SPLINE
SPL {X  -131.598, Y  +769.376, Z    +0.000, E1   -56.871, E3 +79450.846}
SPL {X  -152.760, Y  +729.846, Z    +0.000, E1   -44.713, E3 +79457.898}
SPL {X  -158.868, Y  +709.157, Z    +0.000, E1   -33.466, E3 +79459.099}
SPL {X  -161.987, Y  +689.949, Z    +0.000, E1   -18.777, E3 +79460.061}
SPL {X  -162.803, Y  +675.860, Z    +0.000, E1    -4.958, E3 +79460.043}
SPL {X  -162.820, Y  +671.500, Z    +0.000, E1    +0.000, E3 +79459.579}
SPL {X  -162.820, Y  +669.410, Z    +0.000, E1    +4.515, E3 +79459.341}
SPL {X  -162.820, Y  +664.781, Z    +0.000, E1   +16.411, E3 +79459.337}
SPL {X  -162.820, Y  +659.650, Z    +0.000, E1   +29.778, E3 +79459.346}
SPL {X  -162.820, Y  +654.031, Z    +0.000, E1   +42.449, E3 +79459.260}
SPL {X  -162.820, Y  +647.611, Z    +0.000, E1   +52.483, E3 +79459.791}
SPL {X  -162.820, Y  +637.134, Z    +0.000, E1   +65.232, E3 +79458.039}
SPL {X  -162.820, Y  +616.721, Z    +0.000, E1   +72.273, E3 +79461.773}
SPL {X  -162.820, Y  +577.172, Z    +0.000, E1   +75.843, E3 +79471.753}
SPL {X  -159.895, Y  +349.775, Z    +0.000, E1   +76.042, E3 +79563.419}
ENDSPLINE

SPLINE
SPL {X  -160.357, Y  +352.285, Z    +0.000, E1   +74.783, E3 +79576.357}
ENDSPLINE

SPLINE
SPL {X  -145.737, Y  +307.897, Z    +0.000, E1   +77.368, E3 +79568.932}
SPL {X  -145.329, Y  +307.084, Z    +0.000, E1   +76.571, E3 +79577.768}
ENDSPLINE

SPLINE
SPL {X  -145.355, Y  +307.136, Z    +0.000, E1   +75.607, E3 +79587.292}
ENDSPLINE

SPLINE
SPL {X  -144.515, Y  +305.495, Z    +0.000, E1   +74.543, E3 +79598.101}
SPL {X  -143.690, Y  +303.925, Z    +0.000, E1   +73.372, E3 +79608.840}
SPL {X  -141.993, Y  +300.823, Z    +0.000, E1   +72.659, E3 +79616.265}
SPL {X  -138.166, Y  +294.358, Z    +0.000, E1   +72.281, E3 +79622.726}
SPL {X  -134.385, Y  +288.571, Z    +0.000, E1   +71.826, E3 +79628.990}
SPL {X  -130.773, Y  +283.501, Z    +0.000, E1   +71.398, E3 +79634.414}
SPL {X  -126.922, Y  +278.513, Z    +0.000, E1   +70.767, E3 +79640.568}
SPL {X  -123.520, Y  +274.419, Z    +0.000, E1   +70.342, E3 +79644.767}
SPL {X  -117.513, Y  +267.801, Z    +0.000, E1   +72.197, E3 +79641.115}
SPL {X   -63.140, Y  +230.421, Z    +0.000, E1   +55.875, E3 +79810.554}
ENDSPLINE

SPLINE
SPL {X  -130.329, Y  +282.905, Z    +0.000, E1   +55.659, E3 +79968.890}
SPL {X  -154.728, Y  +329.807, Z    +0.000, E1   +40.640, E3 +79978.271}
SPL {X  -160.994, Y  +356.185, Z    +0.000, E1   +24.373, E3 +79980.864}
SPL {X  -162.637, Y  +372.778, Z    +0.000, E1   +10.098, E3 +79980.884}
SPL {X  -162.820, Y  +382.419, Z    +0.000, E1    +0.163, E3 +79980.444}
SPL {X  -162.820, Y  +383.794, Z    +0.000, E1    -2.626, E3 +79980.162}
SPL {X  -162.820, Y  +387.647, Z    +0.000, E1   -11.488, E3 +79980.166}
SPL {X  -162.820, Y  +394.732, Z    +0.000, E1   -28.992, E3 +79980.084}
SPL {X  -162.820, Y  +403.075, Z    +0.000, E1   -46.096, E3 +79980.314}
SPL {X  -162.820, Y  +414.705, Z    +0.000, E1   -61.052, E3 +79979.760}
SPL {X  -162.820, Y  +466.149, Z    +0.000, E1   -74.732, E3 +79989.756}
SPL {X  -160.066, Y  +703.318, Z    +0.000, E1   -76.774, E3 +80074.603}
ENDSPLINE

SPLINE
SPL {X  -161.105, Y  +697.069, Z    +0.000, E1   -74.557, E3 +80096.218}
ENDSPLINE

SPLINE
SPL {X  -159.270, Y  +707.314, Z    +0.000, E1   -74.359, E3 +80104.241}
SPL {X  -156.868, Y  +717.123, Z    +0.000, E1   -74.182, E3 +80111.747}
SPL {X  -153.226, Y  +728.564, Z    +0.000, E1   -73.755, E3 +80122.756}
SPL {X  -149.090, Y  +738.941, Z    +0.000, E1   -73.348, E3 +80132.329}
SPL {X  -145.714, Y  +746.149, Z    +0.000, E1   -72.951, E3 +80139.916}
SPL {X  -142.592, Y  +752.100, Z    +0.000, E1   -72.554, E3 +80146.449}
SPL {X  -139.608, Y  +757.285, Z    +0.000, E1   -72.326, E3 +80151.118}
SPL {X  -136.902, Y  +761.638, Z    +0.000, E1   -71.857, E3 +80156.886}
SPL {X  -133.350, Y  +766.925, Z    +0.000, E1   -71.498, E3 +80162.206}
SPL {X  -129.687, Y  +771.946, Z    +0.000, E1   -71.061, E3 +80167.572}
SPL {X  -126.374, Y  +776.164, Z    +0.000, E1   -70.494, E3 +80172.826}
SPL {X  -123.763, Y  +779.297, Z    +0.000, E1   -70.128, E3 +80176.201}
SPL {X  -119.350, Y  +784.252, Z    +0.000, E1   -71.016, E3 +80175.402}
SPL {X   -61.593, Y  +824.220, Z    +0.000, E1   -55.970, E3 +80341.717}
ENDSPLINE

SPLINE
SPL {X  -131.598, Y  +769.376, Z    +0.000, E1   -56.871, E3 +80507.989}
SPL {X  -152.760, Y  +729.846, Z    +0.000, E1   -44.713, E3 +80515.041}
SPL {X  -159.952, Y  +703.925, Z    +0.000, E1   -29.977, E3 +80516.544}
SPL {X  -162.596, Y  +682.036, Z    +0.000, E1   -11.376, E3 +80517.264}
SPL {X  -162.820, Y  +671.380, Z    +0.000, E1    +0.035, E3 +80516.703}
SPL {X  -162.820, Y  +668.318, Z    +0.000, E1    +7.404, E3 +80516.440}
SPL {X  -162.820, Y  +664.781, Z    +0.000, E1   +16.411, E3 +80516.480}
SPL {X  -162.820, Y  +659.650, Z    +0.000, E1   +29.778, E3 +80516.489}
SPL {X  -162.820, Y  +651.175, Z    +0.000, E1   +47.162, E3 +80516.639}
SPL {X  -162.820, Y  +633.243, Z    +0.000, E1   +67.111, E3 +80515.894}
SPL {X  -162.820, Y  +577.172, Z    +0.000, E1   +75.843, E3 +80528.896}
SPL {X  -159.895, Y  +349.775, Z    +0.000, E1   +76.042, E3 +80620.562}
ENDSPLINE

SPLINE
SPL {X  -160.357, Y  +352.285, Z    +0.000, E1   +74.783, E3 +80633.500}
ENDSPLINE

SPLINE
SPL {X  -145.737, Y  +307.897, Z    +0.000, E1   +77.368, E3 +80626.075}
SPL {X  -145.329, Y  +307.084, Z    +0.000, E1   +76.571, E3 +80634.911}
ENDSPLINE

SPLINE
SPL {X  -145.355, Y  +307.136, Z    +0.000, E1   +75.607, E3 +80644.435}
ENDSPLINE

SPLINE
SPL {X  -144.515, Y  +305.495, Z    +0.000, E1   +74.543, E3 +80655.244}
SPL {X  -143.690, Y  +303.925, Z    +0.000, E1   +73.372, E3 +80665.983}
SPL {X  -141.993, Y  +300.823, Z    +0.000, E1   +72.659, E3 +80673.408}
SPL {X  -138.166, Y  +294.358, Z    +0.000, E1   +72.281, E3 +80679.869}
SPL {X  -134.385, Y  +288.571, Z    +0.000, E1   +71.826, E3 +80686.132}
SPL {X  -130.773, Y  +283.501, Z    +0.000, E1   +71.398, E3 +80691.557}
SPL {X  -126.922, Y  +278.513, Z    +0.000, E1   +70.767, E3 +80697.711}
SPL {X  -123.520, Y  +274.419, Z    +0.000, E1   +70.342, E3 +80701.909}
SPL {X  -117.513, Y  +267.801, Z    +0.000, E1   +72.197, E3 +80698.258}
SPL {X   -63.140, Y  +230.421, Z    +0.000, E1   +55.875, E3 +80867.697}
ENDSPLINE

SPLINE
SPL {X  -130.329, Y  +282.905, Z    +0.000, E1   +55.659, E3 +81026.033}
SPL {X  -150.766, Y  +319.018, Z    +0.000, E1   +45.408, E3 +81034.525}
SPL {X  -157.479, Y  +339.138, Z    +0.000, E1   +35.556, E3 +81035.961}
SPL {X  -160.994, Y  +356.185, Z    +0.000, E1   +24.373, E3 +81038.007}
SPL {X  -162.352, Y  +368.168, Z    +0.000, E1   +14.282, E3 +81038.059}
SPL {X  -162.808, Y  +378.562, Z    +0.000, E1    +4.298, E3 +81037.991}
SPL {X  -162.820, Y  +382.500, Z    +0.000, E1    +0.000, E3 +81037.564}
SPL {X  -162.820, Y  +384.915, Z    +0.000, E1    -4.894, E3 +81037.277}
SPL {X  -162.820, Y  +388.986, Z    +0.000, E1   -15.047, E3 +81037.375}
SPL {X  -162.820, Y  +394.732, Z    +0.000, E1   -28.992, E3 +81037.227}
SPL {X  -162.820, Y  +403.075, Z    +0.000, E1   -46.096, E3 +81037.456}
SPL {X  -162.820, Y  +414.705, Z    +0.000, E1   -61.052, E3 +81036.903}
SPL {X  -162.820, Y  +466.149, Z    +0.000, E1   -74.732, E3 +81046.899}
SPL {X  -160.722, Y  +699.554, Z    +0.000, E1   -75.485, E3 +81144.309}
SPL {X  -159.966, Y  +703.854, Z    +0.000, E1   -74.386, E3 +81159.212}
SPL {X  -156.868, Y  +717.123, Z    +0.000, E1   -74.182, E3 +81168.890}
SPL {X  -153.226, Y  +728.564, Z    +0.000, E1   -73.755, E3 +81179.898}
SPL {X  -149.090, Y  +738.941, Z    +0.000, E1   -73.348, E3 +81189.472}
SPL {X  -145.714, Y  +746.149, Z    +0.000, E1   -72.951, E3 +81197.059}
SPL {X  -140.946, Y  +755.015, Z    +0.000, E1   -72.452, E3 +81206.162}
SPL {X  -136.902, Y  +761.638, Z    +0.000, E1   -71.857, E3 +81214.028}
SPL {X  -133.350, Y  +766.925, Z    +0.000, E1   -71.498, E3 +81219.349}
SPL {X  -129.687, Y  +771.946, Z    +0.000, E1   -71.061, E3 +81224.715}
SPL {X  -126.374, Y  +776.164, Z    +0.000, E1   -70.494, E3 +81229.968}
SPL {X  -122.717, Y  +780.508, Z    +0.000, E1   -70.361, E3 +81233.006}
SPL {X  -114.093, Y  +789.660, Z    +0.000, E1   -71.634, E3 +81233.024}
SPL {X   -61.593, Y  +824.220, Z    +0.000, E1   -55.970, E3 +81398.860}
ENDSPLINE

SPLINE
SPL {X  -131.598, Y  +769.376, Z    +0.000, E1   -56.871, E3 +81565.132}
SPL {X  -152.760, Y  +729.846, Z    +0.000, E1   -44.713, E3 +81572.184}
SPL {X  -158.868, Y  +709.157, Z    +0.000, E1   -33.466, E3 +81573.385}
SPL {X  -161.987, Y  +689.949, Z    +0.000, E1   -18.777, E3 +81574.346}
SPL {X  -162.803, Y  +675.860, Z    +0.000, E1    -4.958, E3 +81574.328}
SPL {X  -162.820, Y  +671.500, Z    +0.000, E1    +0.000, E3 +81573.865}
SPL {X  -162.820, Y  +669.410, Z    +0.000, E1    +4.515, E3 +81573.627}
SPL {X  -162.820, Y  +664.781, Z    +0.000, E1   +16.411, E3 +81573.622}
SPL {X  -162.820, Y  +659.650, Z    +0.000, E1   +29.778, E3 +81573.632}
SPL {X  -162.820, Y  +651.175, Z    +0.000, E1   +47.162, E3 +81573.782}
SPL {X  -162.820, Y  +637.134, Z    +0.000, E1   +65.232, E3 +81572.324}
SPL {X  -162.820, Y  +616.721, Z    +0.000, E1   +72.273, E3 +81576.058}
SPL {X  -162.820, Y  +577.172, Z    +0.000, E1   +75.843, E3 +81586.039}
SPL {X  -159.895, Y  +349.775, Z    +0.000, E1   +76.042, E3 +81677.705}
ENDSPLINE

SPLINE
SPL {X  -160.357, Y  +352.285, Z    +0.000, E1   +74.783, E3 +81690.642}
ENDSPLINE

SPLINE
SPL {X  -145.737, Y  +307.897, Z    +0.000, E1   +77.368, E3 +81683.218}
SPL {X  -145.329, Y  +307.084, Z    +0.000, E1   +76.571, E3 +81692.054}
ENDSPLINE

SPLINE
SPL {X  -145.355, Y  +307.136, Z    +0.000, E1   +75.607, E3 +81701.578}
ENDSPLINE

SPLINE
SPL {X  -144.515, Y  +305.495, Z    +0.000, E1   +74.543, E3 +81712.387}
SPL {X  -143.690, Y  +303.925, Z    +0.000, E1   +73.372, E3 +81723.126}
SPL {X  -141.993, Y  +300.823, Z    +0.000, E1   +72.659, E3 +81730.551}
SPL {X  -138.166, Y  +294.358, Z    +0.000, E1   +72.281, E3 +81737.012}
SPL {X  -134.385, Y  +288.571, Z    +0.000, E1   +71.826, E3 +81743.275}
SPL {X  -129.872, Y  +282.297, Z    +0.000, E1   +71.229, E3 +81750.445}
SPL {X  -124.448, Y  +275.510, Z    +0.000, E1   +70.509, E3 +81757.818}
SPL {X  -117.513, Y  +267.801, Z    +0.000, E1   +72.197, E3 +81755.401}
SPL {X   -63.140, Y  +230.421, Z    +0.000, E1   +55.875, E3 +81924.840}
ENDSPLINE

SPLINE
SPL {X  -130.329, Y  +282.905, Z    +0.000, E1   +55.659, E3 +82083.176}
SPL {X  -150.766, Y  +319.018, Z    +0.000, E1   +45.408, E3 +82091.668}
SPL {X  -157.479, Y  +339.138, Z    +0.000, E1   +35.556, E3 +82093.104}
SPL {X  -160.994, Y  +356.185, Z    +0.000, E1   +24.373, E3 +82095.150}
SPL {X  -162.352, Y  +368.168, Z    +0.000, E1   +14.282, E3 +82095.202}
SPL {X  -162.808, Y  +378.562, Z    +0.000, E1    +4.298, E3 +82095.134}
SPL {X  -162.820, Y  +382.500, Z    +0.000, E1    +0.000, E3 +82094.707}
SPL {X  -162.820, Y  +383.794, Z    +0.000, E1    -2.626, E3 +82094.448}
SPL {X  -162.820, Y  +387.647, Z    +0.000, E1   -11.488, E3 +82094.451}
SPL {X  -162.820, Y  +393.007, Z    +0.000, E1   -25.093, E3 +82094.409}
SPL {X  -162.820, Y  +400.636, Z    +0.000, E1   -41.711, E3 +82094.459}
SPL {X  -162.820, Y  +414.705, Z    +0.000, E1   -61.052, E3 +82094.046}
SPL {X  -162.820, Y  +466.149, Z    +0.000, E1   -74.732, E3 +82104.042}
SPL {X  -160.066, Y  +703.318, Z    +0.000, E1   -76.774, E3 +82188.889}
ENDSPLINE

SPLINE
SPL {X  -161.105, Y  +697.069, Z    +0.000, E1   -74.557, E3 +82210.503}
ENDSPLINE

SPLINE
SPL {X  -159.270, Y  +707.314, Z    +0.000, E1   -74.359, E3 +82218.527}
SPL {X  -156.868, Y  +717.123, Z    +0.000, E1   -74.182, E3 +82226.033}
SPL {X  -153.226, Y  +728.564, Z    +0.000, E1   -73.755, E3 +82237.041}
SPL {X  -149.090, Y  +738.941, Z    +0.000, E1   -73.348, E3 +82246.615}
SPL {X  -145.714, Y  +746.149, Z    +0.000, E1   -72.951, E3 +82254.202}
SPL {X  -140.946, Y  +755.015, Z    +0.000, E1   -72.452, E3 +82263.305}
SPL {X  -136.902, Y  +761.638, Z    +0.000, E1   -71.857, E3 +82271.171}
SPL {X  -133.350, Y  +766.925, Z    +0.000, E1   -71.498, E3 +82276.492}
SPL {X  -129.687, Y  +771.946, Z    +0.000, E1   -71.061, E3 +82281.858}
SPL {X  -126.374, Y  +776.164, Z    +0.000, E1   -70.494, E3 +82287.111}
SPL {X  -123.763, Y  +779.297, Z    +0.000, E1   -70.128, E3 +82290.487}
SPL {X  -119.350, Y  +784.252, Z    +0.000, E1   -71.016, E3 +82289.687}
SPL {X   -61.593, Y  +824.220, Z    +0.000, E1   -55.970, E3 +82456.003}
ENDSPLINE

SPLINE
SPL {X  -131.598, Y  +769.376, Z    +0.000, E1   -56.871, E3 +82622.275}
SPL {X  -152.760, Y  +729.846, Z    +0.000, E1   -44.713, E3 +82629.327}
SPL {X  -158.868, Y  +709.157, Z    +0.000, E1   -33.466, E3 +82630.528}
SPL {X  -161.987, Y  +689.949, Z    +0.000, E1   -18.777, E3 +82631.489}
SPL {X  -162.803, Y  +675.860, Z    +0.000, E1    -4.958, E3 +82631.471}
SPL {X  -162.820, Y  +671.500, Z    +0.000, E1    +0.000, E3 +82631.008}
SPL {X  -162.820, Y  +669.410, Z    +0.000, E1    +4.515, E3 +82630.770}
SPL {X  -162.820, Y  +664.781, Z    +0.000, E1   +16.411, E3 +82630.765}
SPL {X  -162.820, Y  +659.650, Z    +0.000, E1   +29.778, E3 +82630.775}
SPL {X  -162.820, Y  +651.175, Z    +0.000, E1   +47.162, E3 +82630.925}
SPL {X  -162.820, Y  +633.243, Z    +0.000, E1   +67.111, E3 +82630.180}
SPL {X  -162.820, Y  +577.172, Z    +0.000, E1   +75.843, E3 +82643.181}
SPL {X  -159.895, Y  +349.775, Z    +0.000, E1   +76.042, E3 +82734.848}
ENDSPLINE

SPLINE
SPL {X  -160.357, Y  +352.285, Z    +0.000, E1   +74.783, E3 +82747.785}
ENDSPLINE

SPLINE
SPL {X  -145.737, Y  +307.897, Z    +0.000, E1   +77.368, E3 +82740.361}
SPL {X  -145.329, Y  +307.084, Z    +0.000, E1   +76.571, E3 +82749.197}
ENDSPLINE

SPLINE
SPL {X  -145.355, Y  +307.136, Z    +0.000, E1   +75.607, E3 +82758.721}
ENDSPLINE

SPLINE
SPL {X  -144.841, Y  +306.126, Z    +0.000, E1   +74.709, E3 +82767.595}
SPL {X  -143.742, Y  +304.025, Z    +0.000, E1   +73.644, E3 +82778.121}
SPL {X  -141.993, Y  +300.823, Z    +0.000, E1   +72.659, E3 +82787.693}
SPL {X  -138.166, Y  +294.358, Z    +0.000, E1   +72.281, E3 +82794.155}
SPL {X  -134.385, Y  +288.571, Z    +0.000, E1   +71.826, E3 +82800.418}
SPL {X  -130.773, Y  +283.501, Z    +0.000, E1   +71.398, E3 +82805.842}
SPL {X  -126.922, Y  +278.513, Z    +0.000, E1   +70.767, E3 +82811.996}
SPL {X  -123.520, Y  +274.419, Z    +0.000, E1   +70.342, E3 +82816.195}
SPL {X  -117.513, Y  +267.801, Z    +0.000, E1   +72.197, E3 +82812.544}
SPL {X   -63.140, Y  +230.421, Z    +0.000, E1   +55.875, E3 +82981.983}
ENDSPLINE

SPLINE
SPL {X  -130.329, Y  +282.905, Z    +0.000, E1   +55.659, E3 +83140.318}
SPL {X  -154.728, Y  +329.807, Z    +0.000, E1   +40.640, E3 +83149.700}
SPL {X  -160.994, Y  +356.185, Z    +0.000, E1   +24.373, E3 +83152.293}
SPL {X  -162.352, Y  +368.168, Z    +0.000, E1   +14.282, E3 +83152.345}
SPL {X  -162.808, Y  +378.562, Z    +0.000, E1    +4.298, E3 +83152.277}
SPL {X  -162.820, Y  +382.822, Z    +0.000, E1    -0.352, E3 +83151.785}
SPL {X  -162.820, Y  +387.647, Z    +0.000, E1   -11.488, E3 +83151.594}
SPL {X  -162.820, Y  +393.007, Z    +0.000, E1   -25.093, E3 +83151.552}
SPL {X  -162.820, Y  +400.636, Z    +0.000, E1   -41.711, E3 +83151.602}
SPL {X  -162.820, Y  +414.705, Z    +0.000, E1   -61.052, E3 +83151.188}
SPL {X  -162.820, Y  +466.149, Z    +0.000, E1   -74.732, E3 +83161.185}
SPL {X  -160.066, Y  +703.318, Z    +0.000, E1   -76.774, E3 +83246.032}
ENDSPLINE

SPLINE
SPL {X  -161.105, Y  +697.069, Z    +0.000, E1   -74.557, E3 +83267.646}
ENDSPLINE

SPLINE
SPL {X  -159.270, Y  +707.314, Z    +0.000, E1   -74.359, E3 +83275.670}
SPL {X  -156.868, Y  +717.123, Z    +0.000, E1   -74.182, E3 +83283.176}
SPL {X  -154.373, Y  +725.261, Z    +0.000, E1   -73.879, E3 +83290.886}
SPL {X  -152.060, Y  +731.708, Z    +0.000, E1   -73.572, E3 +83297.534}
SPL {X  -149.090, Y  +738.941, Z    +0.000, E1   -73.348, E3 +83303.758}
SPL {X  -145.714, Y  +746.149, Z    +0.000, E1   -72.951, E3 +83311.345}
SPL {X  -140.946, Y  +755.015, Z    +0.000, E1   -72.452, E3 +83320.447}
SPL {X  -136.902, Y  +761.638, Z    +0.000, E1   -71.857, E3 +83328.314}
SPL {X  -133.350, Y  +766.925, Z    +0.000, E1   -71.498, E3 +83333.635}
SPL {X  -129.687, Y  +771.946, Z    +0.000, E1   -71.061, E3 +83339.001}
SPL {X  -126.374, Y  +776.164, Z    +0.000, E1   -70.494, E3 +83344.254}
SPL {X  -122.717, Y  +780.508, Z    +0.000, E1   -70.361, E3 +83347.292}
SPL {X  -114.093, Y  +789.660, Z    +0.000, E1   -71.634, E3 +83347.310}
SPL {X   -61.795, Y  +824.138, Z    +0.000, E1   -56.629, E3 +83492.977}
ENDSPLINE

SPLINE
SPL {X  -113.687, Y  +790.058, Z    +0.000, E1   -59.721, E3 +83669.724}
SPL {X  -139.151, Y  +758.042, Z    +0.000, E1   -54.091, E3 +83681.284}
SPL {X  -152.760, Y  +729.846, Z    +0.000, E1   -44.713, E3 +83686.470}
SPL {X  -158.868, Y  +709.157, Z    +0.000, E1   -33.466, E3 +83687.671}
SPL {X  -161.987, Y  +689.949, Z    +0.000, E1   -18.777, E3 +83688.632}
SPL {X  -162.743, Y  +678.515, Z    +0.000, E1    -7.658, E3 +83688.627}
SPL {X  -162.820, Y  +671.380, Z    +0.000, E1    +0.035, E3 +83688.132}
SPL {X  -162.820, Y  +668.318, Z    +0.000, E1    +7.404, E3 +83687.869}
SPL {X  -162.820, Y  +664.781, Z    +0.000, E1   +16.411, E3 +83687.908}
SPL {X  -162.820, Y  +659.650, Z    +0.000, E1   +29.778, E3 +83687.918}
SPL {X  -162.820, Y  +651.175, Z    +0.000, E1   +47.162, E3 +83688.068}
SPL {X  -162.820, Y  +633.243, Z    +0.000, E1   +67.111, E3 +83687.323}
SPL {X  -162.820, Y  +577.172, Z    +0.000, E1   +75.843, E3 +83700.324}
SPL {X  -159.895, Y  +349.775, Z    +0.000, E1   +76.042, E3 +83791.990}
ENDSPLINE

SPLINE
SPL {X  -160.357, Y  +352.285, Z    +0.000, E1   +74.783, E3 +83804.928}
ENDSPLINE

SPLINE
SPL {X  -145.737, Y  +307.897, Z    +0.000, E1   +77.368, E3 +83797.503}
SPL {X  -145.329, Y  +307.084, Z    +0.000, E1   +76.571, E3 +83806.340}
ENDSPLINE

SPLINE
SPL {X  -145.355, Y  +307.136, Z    +0.000, E1   +75.607, E3 +83815.864}
ENDSPLINE

SPLINE
SPL {X  -144.515, Y  +305.495, Z    +0.000, E1   +74.543, E3 +83826.673}
SPL {X  -143.690, Y  +303.925, Z    +0.000, E1   +73.372, E3 +83837.412}
SPL {X  -141.993, Y  +300.823, Z    +0.000, E1   +72.659, E3 +83844.836}
SPL {X  -138.166, Y  +294.358, Z    +0.000, E1   +72.281, E3 +83851.297}
SPL {X  -134.385, Y  +288.571, Z    +0.000, E1   +71.826, E3 +83857.561}
SPL {X  -129.872, Y  +282.297, Z    +0.000, E1   +71.229, E3 +83864.731}
SPL {X  -124.448, Y  +275.510, Z    +0.000, E1   +70.509, E3 +83872.104}
SPL {X  -117.513, Y  +267.801, Z    +0.000, E1   +72.197, E3 +83869.687}
SPL {X   -63.140, Y  +230.421, Z    +0.000, E1   +55.875, E3 +84039.125}
ENDSPLINE

SPLINE
SPL {X  -130.329, Y  +282.905, Z    +0.000, E1   +55.659, E3 +84197.461}
SPL {X  -154.728, Y  +329.807, Z    +0.000, E1   +40.640, E3 +84206.843}
SPL {X  -160.994, Y  +356.185, Z    +0.000, E1   +24.373, E3 +84209.435}
SPL {X  -162.637, Y  +372.778, Z    +0.000, E1   +10.098, E3 +84209.456}
SPL {X  -162.820, Y  +382.748, Z    +0.000, E1    -0.178, E3 +84208.948}
SPL {X  -162.820, Y  +387.647, Z    +0.000, E1   -11.488, E3 +84208.737}
SPL {X  -162.820, Y  +393.007, Z    +0.000, E1   -25.093, E3 +84208.695}
SPL {X  -162.820, Y  +400.636, Z    +0.000, E1   -41.711, E3 +84208.745}
SPL {X  -162.820, Y  +414.705, Z    +0.000, E1   -61.052, E3 +84208.331}
SPL {X  -162.820, Y  +466.149, Z    +0.000, E1   -74.732, E3 +84218.327}
SPL {X  -160.722, Y  +699.554, Z    +0.000, E1   -75.485, E3 +84315.737}
SPL {X  -159.966, Y  +703.854, Z    +0.000, E1   -74.386, E3 +84330.641}
SPL {X  -156.868, Y  +717.123, Z    +0.000, E1   -74.182, E3 +84340.319}
SPL {X  -153.226, Y  +728.564, Z    +0.000, E1   -73.755, E3 +84351.327}
SPL {X  -149.090, Y  +738.941, Z    +0.000, E1   -73.348, E3 +84360.901}
SPL {X  -145.714, Y  +746.149, Z    +0.000, E1   -72.951, E3 +84368.487}
SPL {X  -140.946, Y  +755.015, Z    +0.000, E1   -72.452, E3 +84377.590}
SPL {X  -136.902, Y  +761.638, Z    +0.000, E1   -71.857, E3 +84385.457}
SPL {X  -133.350, Y  +766.925, Z    +0.000, E1   -71.498, E3 +84390.778}
SPL {X  -129.687, Y  +771.946, Z    +0.000, E1   -71.061, E3 +84396.144}
SPL {X  -126.374, Y  +776.164, Z    +0.000, E1   -70.494, E3 +84401.397}
SPL {X  -123.763, Y  +779.297, Z    +0.000, E1   -70.128, E3 +84404.773}
SPL {X  -119.350, Y  +784.252, Z    +0.000, E1   -71.016, E3 +84403.973}
SPL {X   -61.593, Y  +824.220, Z    +0.000, E1   -55.970, E3 +84570.289}
ENDSPLINE

SPLINE
SPL {X  -131.598, Y  +769.376, Z    +0.000, E1   -56.871, E3 +84736.560}
SPL {X  -152.760, Y  +729.846, Z    +0.000, E1   -44.713, E3 +84743.613}
SPL {X  -158.868, Y  +709.157, Z    +0.000, E1   -33.466, E3 +84744.814}
SPL {X  -161.987, Y  +689.949, Z    +0.000, E1   -18.777, E3 +84745.775}
SPL {X  -162.803, Y  +675.860, Z    +0.000, E1    -4.958, E3 +84745.757}
SPL {X  -162.820, Y  +671.500, Z    +0.000, E1    +0.000, E3 +84745.293}
SPL {X  -162.820, Y  +669.410, Z    +0.000, E1    +4.515, E3 +84745.056}
SPL {X  -162.820, Y  +664.781, Z    +0.000, E1   +16.411, E3 +84745.051}
SPL {X  -162.820, Y  +659.650, Z    +0.000, E1   +29.778, E3 +84745.061}
SPL {X  -162.820, Y  +654.031, Z    +0.000, E1   +42.449, E3 +84744.975}
SPL {X  -162.820, Y  +647.611, Z    +0.000, E1   +52.483, E3 +84745.505}
SPL {X  -162.820, Y  +633.243, Z    +0.000, E1   +67.111, E3 +84744.465}
SPL {X  -162.820, Y  +577.172, Z    +0.000, E1   +75.843, E3 +84757.467}
SPL {X  -159.895, Y  +349.775, Z    +0.000, E1   +76.042, E3 +84849.133}
ENDSPLINE

SPLINE
SPL {X  -160.357, Y  +352.285, Z    +0.000, E1   +74.783, E3 +84862.071}
ENDSPLINE

SPLINE
SPL {X  -145.737, Y  +307.897, Z    +0.000, E1   +77.368, E3 +84854.646}
SPL {X  -145.329, Y  +307.084, Z    +0.000, E1   +76.571, E3 +84863.482}
ENDSPLINE

SPLINE
SPL {X  -145.355, Y  +307.136, Z    +0.000, E1   +75.607, E3 +84873.007}
ENDSPLINE

SPLINE
SPL {X  -144.515, Y  +305.495, Z    +0.000, E1   +74.543, E3 +84883.816}
SPL {X  -143.690, Y  +303.925, Z    +0.000, E1   +73.372, E3 +84894.554}
SPL {X  -141.993, Y  +300.823, Z    +0.000, E1   +72.659, E3 +84901.979}
SPL {X  -138.166, Y  +294.358, Z    +0.000, E1   +72.281, E3 +84908.440}
SPL {X  -134.385, Y  +288.571, Z    +0.000, E1   +71.826, E3 +84914.704}
SPL {X  -130.773, Y  +283.501, Z    +0.000, E1   +71.398, E3 +84920.128}
SPL {X  -126.922, Y  +278.513, Z    +0.000, E1   +70.767, E3 +84926.282}
SPL {X  -123.520, Y  +274.419, Z    +0.000, E1   +70.342, E3 +84930.481}
SPL {X  -117.513, Y  +267.801, Z    +0.000, E1   +72.197, E3 +84926.830}
SPL {X   -63.140, Y  +230.421, Z    +0.000, E1   +55.875, E3 +85096.268}
ENDSPLINE

SPLINE
SPL {X  -130.329, Y  +282.905, Z    +0.000, E1   +55.659, E3 +85254.604}
SPL {X  -154.728, Y  +329.807, Z    +0.000, E1   +40.640, E3 +85263.985}
SPL {X  -160.994, Y  +356.185, Z    +0.000, E1   +24.373, E3 +85266.578}
SPL {X  -162.352, Y  +368.168, Z    +0.000, E1   +14.282, E3 +85266.631}
SPL {X  -162.808, Y  +378.562, Z    +0.000, E1    +4.298, E3 +85266.563}
SPL {X  -162.820, Y  +382.500, Z    +0.000, E1    +0.000, E3 +85266.136}
SPL {X  -162.820, Y  +384.915, Z    +0.000, E1    -4.894, E3 +85265.849}
SPL {X  -162.820, Y  +388.986, Z    +0.000, E1   -15.047, E3 +85265.947}
SPL {X  -162.820, Y  +393.007, Z    +0.000, E1   -25.093, E3 +85265.838}
SPL {X  -162.820, Y  +400.636, Z    +0.000, E1   -41.711, E3 +85265.888}
SPL {X  -162.820, Y  +414.705, Z    +0.000, E1   -61.052, E3 +85265.474}
SPL {X  -162.820, Y  +466.149, Z    +0.000, E1   -74.732, E3 +85275.470}
SPL {X  -160.066, Y  +703.318, Z    +0.000, E1   -76.774, E3 +85360.318}
ENDSPLINE

SPLINE
SPL {X  -161.105, Y  +697.069, Z    +0.000, E1   -74.557, E3 +85381.932}
ENDSPLINE

SPLINE
SPL {X  -159.270, Y  +707.314, Z    +0.000, E1   -74.359, E3 +85389.956}
SPL {X  -156.868, Y  +717.123, Z    +0.000, E1   -74.182, E3 +85397.462}
SPL {X  -153.226, Y  +728.564, Z    +0.000, E1   -73.755, E3 +85408.470}
SPL {X  -149.090, Y  +738.941, Z    +0.000, E1   -73.348, E3 +85418.043}
SPL {X  -145.714, Y  +746.149, Z    +0.000, E1   -72.951, E3 +85425.630}
SPL {X  -140.946, Y  +755.015, Z    +0.000, E1   -72.452, E3 +85434.733}
SPL {X  -136.902, Y  +761.638, Z    +0.000, E1   -71.857, E3 +85442.600}
SPL {X  -133.350, Y  +766.925, Z    +0.000, E1   -71.498, E3 +85447.920}
SPL {X  -129.687, Y  +771.946, Z    +0.000, E1   -71.061, E3 +85453.286}
SPL {X  -126.374, Y  +776.164, Z    +0.000, E1   -70.494, E3 +85458.540}
SPL {X  -122.717, Y  +780.508, Z    +0.000, E1   -70.361, E3 +85461.577}
SPL {X  -114.093, Y  +789.660, Z    +0.000, E1   -71.634, E3 +85461.596}
SPL {X   -61.593, Y  +824.220, Z    +0.000, E1   -55.970, E3 +85627.431}
ENDSPLINE

SPLINE
SPL {X  -131.598, Y  +769.376, Z    +0.000, E1   -56.871, E3 +85793.703}
SPL {X  -152.760, Y  +729.846, Z    +0.000, E1   -44.713, E3 +85800.756}
SPL {X  -158.868, Y  +709.157, Z    +0.000, E1   -33.466, E3 +85801.957}
SPL {X  -161.987, Y  +689.949, Z    +0.000, E1   -18.777, E3 +85802.918}
SPL {X  -162.803, Y  +675.860, Z    +0.000, E1    -4.958, E3 +85802.900}
SPL {X  -162.820, Y  +671.500, Z    +0.000, E1    +0.000, E3 +85802.436}
SPL {X  -162.820, Y  +669.410, Z    +0.000, E1    +4.515, E3 +85802.198}
SPL {X  -162.820, Y  +664.781, Z    +0.000, E1   +16.411, E3 +85802.194}
SPL {X  -162.820, Y  +659.650, Z    +0.000, E1   +29.778, E3 +85802.204}
SPL {X  -162.820, Y  +654.031, Z    +0.000, E1   +42.449, E3 +85802.117}
SPL {X  -162.820, Y  +647.611, Z    +0.000, E1   +52.483, E3 +85802.648}
SPL {X  -162.820, Y  +633.243, Z    +0.000, E1   +67.111, E3 +85801.608}
SPL {X  -162.820, Y  +577.172, Z    +0.000, E1   +75.843, E3 +85814.610}
SPL {X  -159.895, Y  +349.775, Z    +0.000, E1   +76.042, E3 +85906.276}
ENDSPLINE

SPLINE
SPL {X  -160.357, Y  +352.285, Z    +0.000, E1   +74.783, E3 +85919.214}
ENDSPLINE

SPLINE
SPL {X  -145.737, Y  +307.897, Z    +0.000, E1   +77.368, E3 +85911.789}
SPL {X  -145.329, Y  +307.084, Z    +0.000, E1   +76.571, E3 +85920.625}
ENDSPLINE

SPLINE
SPL {X  -145.355, Y  +307.136, Z    +0.000, E1   +75.607, E3 +85930.149}
ENDSPLINE

SPLINE
SPL {X  -144.515, Y  +305.495, Z    +0.000, E1   +74.543, E3 +85940.959}
SPL {X  -143.690, Y  +303.925, Z    +0.000, E1   +73.372, E3 +85951.697}
SPL {X  -141.993, Y  +300.823, Z    +0.000, E1   +72.659, E3 +85959.122}
SPL {X  -138.166, Y  +294.358, Z    +0.000, E1   +72.281, E3 +85965.583}
SPL {X  -134.385, Y  +288.571, Z    +0.000, E1   +71.826, E3 +85971.847}
SPL {X  -129.872, Y  +282.297, Z    +0.000, E1   +71.229, E3 +85979.017}
SPL {X  -124.448, Y  +275.510, Z    +0.000, E1   +70.509, E3 +85986.390}
SPL {X  -117.513, Y  +267.801, Z    +0.000, E1   +72.197, E3 +85983.972}
SPL {X   -63.140, Y  +230.421, Z    +0.000, E1   +55.875, E3 +86153.411}
ENDSPLINE

SPLINE
SPL {X  -130.329, Y  +282.905, Z    +0.000, E1   +55.659, E3 +86311.747}
SPL {X  -150.766, Y  +319.018, Z    +0.000, E1   +45.408, E3 +86320.240}
SPL {X  -157.479, Y  +339.138, Z    +0.000, E1   +35.556, E3 +86321.675}
SPL {X  -160.994, Y  +356.185, Z    +0.000, E1   +24.373, E3 +86323.721}
SPL {X  -162.352, Y  +368.168, Z    +0.000, E1   +14.282, E3 +86323.774}
SPL {X  -162.808, Y  +378.562, Z    +0.000, E1    +4.298, E3 +86323.706}
SPL {X  -162.820, Y  +382.500, Z    +0.000, E1    +0.000, E3 +86323.278}
SPL {X  -162.820, Y  +383.794, Z    +0.000, E1    -2.626, E3 +86323.019}
SPL {X  -162.820, Y  +387.647, Z    +0.000, E1   -11.488, E3 +86323.023}
SPL {X  -162.820, Y  +393.007, Z    +0.000, E1   -25.093, E3 +86322.981}
SPL {X  -162.820, Y  +400.636, Z    +0.000, E1   -41.711, E3 +86323.030}
SPL {X  -162.820, Y  +414.705, Z    +0.000, E1   -61.052, E3 +86322.617}
SPL {X  -162.820, Y  +466.149, Z    +0.000, E1   -74.732, E3 +86332.613}
SPL {X  -160.066, Y  +703.318, Z    +0.000, E1   -76.774, E3 +86417.461}
ENDSPLINE

SPLINE
SPL {X  -161.105, Y  +697.069, Z    +0.000, E1   -74.557, E3 +86439.075}
ENDSPLINE

SPLINE
SPL {X  -159.270, Y  +707.314, Z    +0.000, E1   -74.359, E3 +86447.099}
SPL {X  -156.868, Y  +717.123, Z    +0.000, E1   -74.182, E3 +86454.605}
SPL {X  -153.226, Y  +728.564, Z    +0.000, E1   -73.755, E3 +86465.613}
SPL {X  -149.090, Y  +738.941, Z    +0.000, E1   -73.348, E3 +86475.186}
SPL {X  -145.714, Y  +746.149, Z    +0.000, E1   -72.951, E3 +86482.773}
SPL {X  -140.946, Y  +755.015, Z    +0.000, E1   -72.452, E3 +86491.876}
SPL {X  -136.902, Y  +761.638, Z    +0.000, E1   -71.857, E3 +86499.743}
SPL {X  -133.350, Y  +766.925, Z    +0.000, E1   -71.498, E3 +86505.063}
SPL {X  -129.687, Y  +771.946, Z    +0.000, E1   -71.061, E3 +86510.429}
SPL {X  -126.374, Y  +776.164, Z    +0.000, E1   -70.494, E3 +86515.683}
SPL {X  -123.763, Y  +779.297, Z    +0.000, E1   -70.128, E3 +86519.059}
SPL {X  -119.350, Y  +784.252, Z    +0.000, E1   -71.016, E3 +86518.259}
SPL {X   -61.593, Y  +824.220, Z    +0.000, E1   -55.970, E3 +86684.574}
ENDSPLINE

SPLINE
SPL {X  -131.598, Y  +769.376, Z    +0.000, E1   -56.871, E3 +86850.846}
SPL {X  -152.760, Y  +729.846, Z    +0.000, E1   -44.713, E3 +86857.898}
SPL {X  -158.868, Y  +709.157, Z    +0.000, E1   -33.466, E3 +86859.099}
SPL {X  -161.987, Y  +689.949, Z    +0.000, E1   -18.777, E3 +86860.061}
SPL {X  -162.743, Y  +678.515, Z    +0.000, E1    -7.658, E3 +86860.056}
SPL {X  -162.820, Y  +671.588, Z    +0.000, E1    -0.190, E3 +86859.602}
SPL {X  -162.820, Y  +669.410, Z    +0.000, E1    +4.515, E3 +86859.341}
SPL {X  -162.820, Y  +664.781, Z    +0.000, E1   +16.411, E3 +86859.337}
SPL {X  -162.820, Y  +659.650, Z    +0.000, E1   +29.778, E3 +86859.346}
SPL {X  -162.820, Y  +654.031, Z    +0.000, E1   +42.449, E3 +86859.260}
SPL {X  -162.820, Y  +647.611, Z    +0.000, E1   +52.483, E3 +86859.791}
SPL {X  -162.820, Y  +637.134, Z    +0.000, E1   +65.232, E3 +86858.039}
SPL {X  -162.820, Y  +616.721, Z    +0.000, E1   +72.273, E3 +86861.773}
SPL {X  -162.820, Y  +577.172, Z    +0.000, E1   +75.843, E3 +86871.753}
SPL {X  -159.895, Y  +349.775, Z    +0.000, E1   +76.042, E3 +86963.419}
ENDSPLINE

SPLINE
SPL {X  -160.357, Y  +352.285, Z    +0.000, E1   +74.783, E3 +86976.357}
ENDSPLINE

SPLINE
SPL {X  -145.737, Y  +307.897, Z    +0.000, E1   +77.368, E3 +86968.932}
SPL {X  -145.122, Y  +306.676, Z    +0.000, E1   +76.360, E3 +86980.285}
ENDSPLINE

SPLINE
SPL {X  -145.186, Y  +306.802, Z    +0.000, E1   +74.850, E3 +86994.638}
ENDSPLINE

SPLINE
SPL {X  -143.742, Y  +304.025, Z    +0.000, E1   +73.644, E3 +87006.692}
SPL {X  -141.993, Y  +300.823, Z    +0.000, E1   +72.659, E3 +87016.265}
SPL {X  -138.166, Y  +294.358, Z    +0.000, E1   +72.281, E3 +87022.726}
SPL {X  -134.385, Y  +288.571, Z    +0.000, E1   +71.826, E3 +87028.990}
SPL {X  -129.872, Y  +282.297, Z    +0.000, E1   +71.229, E3 +87036.160}
SPL {X  -124.448, Y  +275.510, Z    +0.000, E1   +70.509, E3 +87043.533}
SPL {X  -117.513, Y  +267.801, Z    +0.000, E1   +72.197, E3 +87041.115}
SPL {X   -63.140, Y  +230.421, Z    +0.000, E1   +55.875, E3 +87210.554}
ENDSPLINE

SPLINE
SPL {X  -130.329, Y  +282.905, Z    +0.000, E1   +55.659, E3 +87368.890}
SPL {X  -150.766, Y  +319.018, Z    +0.000, E1   +45.408, E3 +87377.383}
SPL {X  -157.479, Y  +339.138, Z    +0.000, E1   +35.556, E3 +87378.818}
SPL {X  -160.994, Y  +356.185, Z    +0.000, E1   +24.373, E3 +87380.864}
SPL {X  -162.352, Y  +368.168, Z    +0.000, E1   +14.282, E3 +87380.917}
SPL {X  -162.808, Y  +378.562, Z    +0.000, E1    +4.298, E3 +87380.848}
SPL {X  -162.820, Y  +382.500, Z    +0.000, E1    +0.000, E3 +87380.421}
SPL {X  -162.820, Y  +383.794, Z    +0.000, E1    -2.626, E3 +87380.162}
SPL {X  -162.820, Y  +387.647, Z    +0.000, E1   -11.488, E3 +87380.166}
SPL {X  -162.820, Y  +393.007, Z    +0.000, E1   -25.093, E3 +87380.124}
SPL {X  -162.820, Y  +400.636, Z    +0.000, E1   -41.711, E3 +87380.173}
SPL {X  -162.820, Y  +414.705, Z    +0.000, E1   -61.052, E3 +87379.760}
SPL {X  -162.820, Y  +466.149, Z    +0.000, E1   -74.732, E3 +87389.756}
SPL {X  -160.722, Y  +699.554, Z    +0.000, E1   -75.485, E3 +87487.166}
SPL {X  -159.966, Y  +703.854, Z    +0.000, E1   -74.386, E3 +87502.069}
SPL {X  -156.868, Y  +717.123, Z    +0.000, E1   -74.182, E3 +87511.747}
SPL {X  -154.373, Y  +725.261, Z    +0.000, E1   -73.879, E3 +87519.457}
SPL {X  -152.060, Y  +731.708, Z    +0.000, E1   -73.572, E3 +87526.105}
SPL {X  -149.090, Y  +738.941, Z    +0.000, E1   -73.348, E3 +87532.329}
SPL {X  -145.714, Y  +746.149, Z    +0.000, E1   -72.951, E3 +87539.916}
SPL {X  -140.946, Y  +755.015, Z    +0.000, E1   -72.452, E3 +87549.019}
SPL {X  -136.902, Y  +761.638, Z    +0.000, E1   -71.857, E3 +87556.886}
SPL {X  -133.350, Y  +766.925, Z    +0.000, E1   -71.498, E3 +87562.206}
SPL {X  -129.687, Y  +771.946, Z    +0.000, E1   -71.061, E3 +87567.572}
SPL {X  -126.374, Y  +776.164, Z    +0.000, E1   -70.494, E3 +87572.826}
SPL {X  -122.717, Y  +780.508, Z    +0.000, E1   -70.361, E3 +87575.863}
SPL {X  -114.093, Y  +789.660, Z    +0.000, E1   -71.634, E3 +87575.881}
SPL {X   -61.795, Y  +824.138, Z    +0.000, E1   -56.629, E3 +87721.549}
ENDSPLINE

SPLINE
SPL {X  -113.687, Y  +790.058, Z    +0.000, E1   -59.721, E3 +87898.296}
SPL {X  -139.151, Y  +758.042, Z    +0.000, E1   -54.091, E3 +87909.855}
SPL {X  -152.760, Y  +729.846, Z    +0.000, E1   -44.713, E3 +87915.041}
SPL {X  -159.952, Y  +703.925, Z    +0.000, E1   -29.977, E3 +87916.544}
SPL {X  -162.596, Y  +682.036, Z    +0.000, E1   -11.376, E3 +87917.264}
SPL {X  -162.820, Y  +671.380, Z    +0.000, E1    +0.035, E3 +87916.703}
SPL {X  -162.820, Y  +668.318, Z    +0.000, E1    +7.404, E3 +87916.440}
SPL {X  -162.820, Y  +664.781, Z    +0.000, E1   +16.411, E3 +87916.480}
SPL {X  -162.820, Y  +659.650, Z    +0.000, E1   +29.778, E3 +87916.489}
SPL {X  -162.820, Y  +651.175, Z    +0.000, E1   +47.162, E3 +87916.639}
SPL {X  -162.820, Y  +633.243, Z    +0.000, E1   +67.111, E3 +87915.894}
SPL {X  -162.820, Y  +577.172, Z    +0.000, E1   +75.843, E3 +87928.896}
SPL {X  -159.895, Y  +349.775, Z    +0.000, E1   +76.042, E3 +88020.562}
ENDSPLINE

SPLINE
SPL {X  -160.357, Y  +352.285, Z    +0.000, E1   +74.783, E3 +88033.500}
ENDSPLINE

SPLINE
SPL {X  -145.737, Y  +307.897, Z    +0.000, E1   +77.368, E3 +88026.075}
SPL {X  -145.329, Y  +307.084, Z    +0.000, E1   +76.571, E3 +88034.911}
ENDSPLINE

SPLINE
SPL {X  -145.355, Y  +307.136, Z    +0.000, E1   +75.607, E3 +88044.435}
ENDSPLINE

SPLINE
SPL {X  -144.841, Y  +306.126, Z    +0.000, E1   +74.709, E3 +88053.309}
SPL {X  -143.742, Y  +304.025, Z    +0.000, E1   +73.644, E3 +88063.835}
SPL {X  -141.993, Y  +300.823, Z    +0.000, E1   +72.659, E3 +88073.408}
SPL {X  -138.166, Y  +294.358, Z    +0.000, E1   +72.281, E3 +88079.869}
SPL {X  -134.385, Y  +288.571, Z    +0.000, E1   +71.826, E3 +88086.132}
SPL {X  -130.773, Y  +283.501, Z    +0.000, E1   +71.398, E3 +88091.557}
SPL {X  -126.922, Y  +278.513, Z    +0.000, E1   +70.767, E3 +88097.711}
SPL {X  -123.520, Y  +274.419, Z    +0.000, E1   +70.342, E3 +88101.909}
SPL {X  -117.513, Y  +267.801, Z    +0.000, E1   +72.197, E3 +88098.258}
SPL {X   -63.140, Y  +230.421, Z    +0.000, E1   +55.875, E3 +88267.697}
ENDSPLINE

SPLINE
SPL {X  -130.329, Y  +282.905, Z    +0.000, E1   +55.659, E3 +88426.033}
SPL {X  -150.766, Y  +319.018, Z    +0.000, E1   +45.408, E3 +88434.525}
SPL {X  -157.479, Y  +339.138, Z    +0.000, E1   +35.556, E3 +88435.961}
SPL {X  -160.994, Y  +356.185, Z    +0.000, E1   +24.373, E3 +88438.007}
SPL {X  -162.637, Y  +372.778, Z    +0.000, E1   +10.098, E3 +88438.027}
SPL {X  -162.820, Y  +382.419, Z    +0.000, E1    +0.163, E3 +88437.587}
SPL {X  -162.820, Y  +384.915, Z    +0.000, E1    -4.894, E3 +88437.277}
SPL {X  -162.820, Y  +388.986, Z    +0.000, E1   -15.047, E3 +88437.375}
SPL {X  -162.820, Y  +393.007, Z    +0.000, E1   -25.093, E3 +88437.266}
SPL {X  -162.820, Y  +400.636, Z    +0.000, E1   -41.711, E3 +88437.316}
SPL {X  -162.820, Y  +414.705, Z    +0.000, E1   -61.052, E3 +88436.903}
SPL {X  -162.820, Y  +466.149, Z    +0.000, E1   -74.732, E3 +88446.899}
SPL {X  -160.066, Y  +703.318, Z    +0.000, E1   -76.774, E3 +88531.746}
ENDSPLINE

SPLINE
SPL {X  -161.105, Y  +697.069, Z    +0.000, E1   -74.557, E3 +88553.361}
ENDSPLINE

SPLINE
SPL {X  -159.270, Y  +707.314, Z    +0.000, E1   -74.359, E3 +88561.384}
SPL {X  -156.868, Y  +717.123, Z    +0.000, E1   -74.182, E3 +88568.890}
SPL {X  -153.226, Y  +728.564, Z    +0.000, E1   -73.755, E3 +88579.898}
SPL {X  -149.090, Y  +738.941, Z    +0.000, E1   -73.348, E3 +88589.472}
SPL {X  -145.714, Y  +746.149, Z    +0.000, E1   -72.951, E3 +88597.059}
SPL {X  -140.946, Y  +755.015, Z    +0.000, E1   -72.452, E3 +88606.162}
SPL {X  -136.902, Y  +761.638, Z    +0.000, E1   -71.857, E3 +88614.028}
SPL {X  -133.350, Y  +766.925, Z    +0.000, E1   -71.498, E3 +88619.349}
SPL {X  -129.687, Y  +771.946, Z    +0.000, E1   -71.061, E3 +88624.715}
SPL {X  -126.374, Y  +776.164, Z    +0.000, E1   -70.494, E3 +88629.968}
SPL {X  -123.763, Y  +779.297, Z    +0.000, E1   -70.128, E3 +88633.344}
SPL {X  -119.350, Y  +784.252, Z    +0.000, E1   -71.016, E3 +88632.544}
SPL {X   -61.593, Y  +824.220, Z    +0.000, E1   -55.970, E3 +88798.860}
ENDSPLINE

SPLINE
SPL {X  -131.598, Y  +769.376, Z    +0.000, E1   -56.871, E3 +88965.132}
SPL {X  -152.760, Y  +729.846, Z    +0.000, E1   -44.713, E3 +88972.184}
SPL {X  -158.868, Y  +709.157, Z    +0.000, E1   -33.466, E3 +88973.385}
SPL {X  -161.987, Y  +689.949, Z    +0.000, E1   -18.777, E3 +88974.346}
SPL {X  -162.803, Y  +675.860, Z    +0.000, E1    -4.958, E3 +88974.328}
SPL {X  -162.820, Y  +671.500, Z    +0.000, E1    +0.000, E3 +88973.865}
SPL {X  -162.820, Y  +669.410, Z    +0.000, E1    +4.515, E3 +88973.627}
SPL {X  -162.820, Y  +664.781, Z    +0.000, E1   +16.411, E3 +88973.622}
SPL {X  -162.820, Y  +659.650, Z    +0.000, E1   +29.778, E3 +88973.632}
SPL {X  -162.820, Y  +651.175, Z    +0.000, E1   +47.162, E3 +88973.782}
SPL {X  -162.820, Y  +633.243, Z    +0.000, E1   +67.111, E3 +88973.037}
SPL {X  -162.820, Y  +577.172, Z    +0.000, E1   +75.843, E3 +88986.039}
SPL {X  -159.895, Y  +349.775, Z    +0.000, E1   +76.042, E3 +89077.705}
ENDSPLINE

SPLINE
SPL {X  -160.357, Y  +352.285, Z    +0.000, E1   +74.783, E3 +89090.642}
ENDSPLINE

SPLINE
SPL {X  -145.737, Y  +307.897, Z    +0.000, E1   +77.368, E3 +89083.218}
SPL {X  -145.329, Y  +307.084, Z    +0.000, E1   +76.571, E3 +89092.054}
ENDSPLINE

SPLINE
SPL {X  -145.355, Y  +307.136, Z    +0.000, E1   +75.607, E3 +89101.578}
ENDSPLINE

SPLINE
SPL {X  -144.515, Y  +305.495, Z    +0.000, E1   +74.543, E3 +89112.387}
SPL {X  -143.690, Y  +303.925, Z    +0.000, E1   +73.372, E3 +89123.126}
SPL {X  -141.993, Y  +300.823, Z    +0.000, E1   +72.659, E3 +89130.551}
SPL {X  -138.166, Y  +294.358, Z    +0.000, E1   +72.281, E3 +89137.012}
SPL {X  -134.385, Y  +288.571, Z    +0.000, E1   +71.826, E3 +89143.275}
SPL {X  -129.872, Y  +282.297, Z    +0.000, E1   +71.229, E3 +89150.445}
SPL {X  -124.448, Y  +275.510, Z    +0.000, E1   +70.509, E3 +89157.818}
SPL {X  -117.513, Y  +267.801, Z    +0.000, E1   +72.197, E3 +89155.401}
SPL {X   -63.140, Y  +230.421, Z    +0.000, E1   +55.875, E3 +89324.840}
ENDSPLINE

SPLINE
SPL {X  -130.329, Y  +282.905, Z    +0.000, E1   +55.659, E3 +89483.176}
SPL {X  -150.766, Y  +319.018, Z    +0.000, E1   +45.408, E3 +89491.668}
SPL {X  -157.479, Y  +339.138, Z    +0.000, E1   +35.556, E3 +89493.104}
SPL {X  -160.994, Y  +356.185, Z    +0.000, E1   +24.373, E3 +89495.150}
SPL {X  -162.637, Y  +372.778, Z    +0.000, E1   +10.098, E3 +89495.170}
SPL {X  -162.820, Y  +382.419, Z    +0.000, E1    +0.163, E3 +89494.730}
SPL {X  -162.820, Y  +384.915, Z    +0.000, E1    -4.894, E3 +89494.420}
SPL {X  -162.820, Y  +388.986, Z    +0.000, E1   -15.047, E3 +89494.518}
SPL {X  -162.820, Y  +393.007, Z    +0.000, E1   -25.093, E3 +89494.409}
SPL {X  -162.820, Y  +400.636, Z    +0.000, E1   -41.711, E3 +89494.459}
SPL {X  -162.820, Y  +414.705, Z    +0.000, E1   -61.052, E3 +89494.046}
SPL {X  -162.820, Y  +466.149, Z    +0.000, E1   -74.732, E3 +89504.042}
SPL {X  -160.722, Y  +699.554, Z    +0.000, E1   -75.485, E3 +89601.452}
SPL {X  -159.966, Y  +703.854, Z    +0.000, E1   -74.386, E3 +89616.355}
SPL {X  -156.868, Y  +717.123, Z    +0.000, E1   -74.182, E3 +89626.033}
SPL {X  -154.373, Y  +725.261, Z    +0.000, E1   -73.879, E3 +89633.743}
SPL {X  -152.060, Y  +731.708, Z    +0.000, E1   -73.572, E3 +89640.391}
SPL {X  -149.090, Y  +738.941, Z    +0.000, E1   -73.348, E3 +89646.615}
SPL {X  -145.714, Y  +746.149, Z    +0.000, E1   -72.951, E3 +89654.202}
SPL {X  -142.592, Y  +752.100, Z    +0.000, E1   -72.554, E3 +89660.734}
SPL {X  -139.608, Y  +757.285, Z    +0.000, E1   -72.326, E3 +89665.404}
SPL {X  -136.902, Y  +761.638, Z    +0.000, E1   -71.857, E3 +89671.171}
SPL {X  -133.350, Y  +766.925, Z    +0.000, E1   -71.498, E3 +89676.492}
SPL {X  -129.687, Y  +771.946, Z    +0.000, E1   -71.061, E3 +89681.858}
SPL {X  -126.374, Y  +776.164, Z    +0.000, E1   -70.494, E3 +89687.111}
SPL {X  -122.717, Y  +780.508, Z    +0.000, E1   -70.361, E3 +89690.149}
SPL {X  -114.093, Y  +789.660, Z    +0.000, E1   -71.634, E3 +89690.167}
SPL {X   -61.795, Y  +824.138, Z    +0.000, E1   -56.629, E3 +89835.834}
ENDSPLINE

SPLINE
SPL {X  -113.687, Y  +790.058, Z    +0.000, E1   -59.721, E3 +90012.582}
SPL {X  -139.151, Y  +758.042, Z    +0.000, E1   -54.091, E3 +90024.141}
SPL {X  -152.760, Y  +729.846, Z    +0.000, E1   -44.713, E3 +90029.327}
SPL {X  -158.868, Y  +709.157, Z    +0.000, E1   -33.466, E3 +90030.528}
SPL {X  -161.987, Y  +689.949, Z    +0.000, E1   -18.777, E3 +90031.489}
SPL {X  -162.743, Y  +678.515, Z    +0.000, E1    -7.658, E3 +90031.484}
SPL {X  -162.820, Y  +671.380, Z    +0.000, E1    +0.035, E3 +90030.989}
SPL {X  -162.820, Y  +668.318, Z    +0.000, E1    +7.404, E3 +90030.726}
SPL {X  -162.820, Y  +664.781, Z    +0.000, E1   +16.411, E3 +90030.765}
SPL {X  -162.820, Y  +659.650, Z    +0.000, E1   +29.778, E3 +90030.775}
SPL {X  -162.820, Y  +651.175, Z    +0.000, E1   +47.162, E3 +90030.925}
SPL {X  -162.820, Y  +633.243, Z    +0.000, E1   +67.111, E3 +90030.180}
SPL {X  -162.820, Y  +577.172, Z    +0.000, E1   +75.843, E3 +90043.181}
SPL {X  -159.895, Y  +349.775, Z    +0.000, E1   +76.042, E3 +90134.848}
ENDSPLINE

SPLINE
SPL {X  -160.357, Y  +352.285, Z    +0.000, E1   +74.783, E3 +90147.785}
ENDSPLINE

SPLINE
SPL {X  -145.737, Y  +307.897, Z    +0.000, E1   +77.368, E3 +90140.361}
SPL {X  -145.329, Y  +307.084, Z    +0.000, E1   +76.571, E3 +90149.197}
ENDSPLINE

SPLINE
SPL {X  -145.355, Y  +307.136, Z    +0.000, E1   +75.607, E3 +90158.721}
ENDSPLINE

SPLINE
SPL {X  -144.515, Y  +305.495, Z    +0.000, E1   +74.543, E3 +90169.530}
SPL {X  -143.690, Y  +303.925, Z    +0.000, E1   +73.372, E3 +90180.269}
SPL {X  -141.993, Y  +300.823, Z    +0.000, E1   +72.659, E3 +90187.693}
SPL {X  -138.166, Y  +294.358, Z    +0.000, E1   +72.281, E3 +90194.155}
SPL {X  -134.385, Y  +288.571, Z    +0.000, E1   +71.826, E3 +90200.418}
SPL {X  -129.872, Y  +282.297, Z    +0.000, E1   +71.229, E3 +90207.588}
SPL {X  -124.448, Y  +275.510, Z    +0.000, E1   +70.509, E3 +90214.961}
SPL {X  -117.513, Y  +267.801, Z    +0.000, E1   +72.197, E3 +90212.544}
SPL {X   -63.140, Y  +230.421, Z    +0.000, E1   +55.875, E3 +90381.983}
ENDSPLINE

SPLINE
SPL {X  -130.329, Y  +282.905, Z    +0.000, E1   +55.659, E3 +90540.318}
SPL {X  -154.728, Y  +329.807, Z    +0.000, E1   +40.640, E3 +90549.700}
SPL {X  -160.994, Y  +356.185, Z    +0.000, E1   +24.373, E3 +90552.293}
SPL {X  -162.637, Y  +372.778, Z    +0.000, E1   +10.098, E3 +90552.313}
SPL {X  -162.820, Y  +382.748, Z    +0.000, E1    -0.178, E3 +90551.805}
SPL {X  -162.820, Y  +387.647, Z    +0.000, E1   -11.488, E3 +90551.594}
SPL {X  -162.820, Y  +393.007, Z    +0.000, E1   -25.093, E3 +90551.552}
SPL {X  -162.820, Y  +400.636, Z    +0.000, E1   -41.711, E3 +90551.602}
SPL {X  -162.820, Y  +414.705, Z    +0.000, E1   -61.052, E3 +90551.188}
SPL {X  -162.820, Y  +466.149, Z    +0.000, E1   -74.732, E3 +90561.185}
SPL {X  -160.722, Y  +699.554, Z    +0.000, E1   -75.485, E3 +90658.595}
SPL {X  -159.966, Y  +703.854, Z    +0.000, E1   -74.386, E3 +90673.498}
SPL {X  -156.868, Y  +717.123, Z    +0.000, E1   -74.182, E3 +90683.176}
SPL {X  -153.226, Y  +728.564, Z    +0.000, E1   -73.755, E3 +90694.184}
SPL {X  -149.090, Y  +738.941, Z    +0.000, E1   -73.348, E3 +90703.758}
SPL {X  -145.714, Y  +746.149, Z    +0.000, E1   -72.951, E3 +90711.345}
SPL {X  -140.946, Y  +755.015, Z    +0.000, E1   -72.452, E3 +90720.447}
SPL {X  -136.902, Y  +761.638, Z    +0.000, E1   -71.857, E3 +90728.314}
SPL {X  -133.350, Y  +766.925, Z    +0.000, E1   -71.498, E3 +90733.635}
SPL {X  -129.687, Y  +771.946, Z    +0.000, E1   -71.061, E3 +90739.001}
SPL {X  -126.374, Y  +776.164, Z    +0.000, E1   -70.494, E3 +90744.254}
SPL {X  -123.763, Y  +779.297, Z    +0.000, E1   -70.128, E3 +90747.630}
SPL {X  -119.350, Y  +784.252, Z    +0.000, E1   -71.016, E3 +90746.830}
SPL {X   -61.593, Y  +824.220, Z    +0.000, E1   -55.970, E3 +90913.146}
ENDSPLINE

SPLINE
SPL {X  -131.598, Y  +769.376, Z    +0.000, E1   -56.871, E3 +91079.418}
SPL {X  -152.760, Y  +729.846, Z    +0.000, E1   -44.713, E3 +91086.470}
SPL {X  -158.868, Y  +709.157, Z    +0.000, E1   -33.466, E3 +91087.671}
SPL {X  -161.987, Y  +689.949, Z    +0.000, E1   -18.777, E3 +91088.632}
SPL {X  -162.803, Y  +675.860, Z    +0.000, E1    -4.958, E3 +91088.614}
SPL {X  -162.820, Y  +671.500, Z    +0.000, E1    +0.000, E3 +91088.151}
SPL {X  -162.820, Y  +669.410, Z    +0.000, E1    +4.515, E3 +91087.913}
SPL {X  -162.820, Y  +664.781, Z    +0.000, E1   +16.411, E3 +91087.908}
SPL {X  -162.820, Y  +659.650, Z    +0.000, E1   +29.778, E3 +91087.918}
SPL {X  -162.820, Y  +654.031, Z    +0.000, E1   +42.449, E3 +91087.832}
SPL {X  -162.820, Y  +647.611, Z    +0.000, E1   +52.483, E3 +91088.362}
SPL {X  -162.820, Y  +633.243, Z    +0.000, E1   +67.111, E3 +91087.323}
SPL {X  -162.820, Y  +577.172, Z    +0.000, E1   +75.843, E3 +91100.324}
SPL {X  -159.895, Y  +349.775, Z    +0.000, E1   +76.042, E3 +91191.990}
ENDSPLINE

SPLINE
SPL {X  -160.357, Y  +352.285, Z    +0.000, E1   +74.783, E3 +91204.928}
ENDSPLINE

SPLINE
SPL {X  -145.737, Y  +307.897, Z    +0.000, E1   +77.368, E3 +91197.503}
SPL {X  -145.329, Y  +307.084, Z    +0.000, E1   +76.571, E3 +91206.340}
ENDSPLINE

SPLINE
SPL {X  -145.355, Y  +307.136, Z    +0.000, E1   +75.607, E3 +91215.864}
ENDSPLINE

SPLINE
SPL {X  -144.515, Y  +305.495, Z    +0.000, E1   +74.543, E3 +91226.673}
SPL {X  -143.690, Y  +303.925, Z    +0.000, E1   +73.372, E3 +91237.412}
SPL {X  -141.993, Y  +300.823, Z    +0.000, E1   +72.659, E3 +91244.836}
SPL {X  -138.166, Y  +294.358, Z    +0.000, E1   +72.281, E3 +91251.297}
SPL {X  -134.385, Y  +288.571, Z    +0.000, E1   +71.826, E3 +91257.561}
SPL {X  -130.773, Y  +283.501, Z    +0.000, E1   +71.398, E3 +91262.985}
SPL {X  -126.922, Y  +278.513, Z    +0.000, E1   +70.767, E3 +91269.139}
SPL {X  -123.520, Y  +274.419, Z    +0.000, E1   +70.342, E3 +91273.338}
SPL {X  -117.513, Y  +267.801, Z    +0.000, E1   +72.197, E3 +91269.687}
SPL {X   -63.140, Y  +230.421, Z    +0.000, E1   +55.875, E3 +91439.125}
ENDSPLINE

SPLINE
SPL {X  -130.329, Y  +282.905, Z    +0.000, E1   +55.659, E3 +91597.461}
SPL {X  -154.728, Y  +329.807, Z    +0.000, E1   +40.640, E3 +91606.843}
SPL {X  -160.994, Y  +356.185, Z    +0.000, E1   +24.373, E3 +91609.435}
SPL {X  -162.352, Y  +368.168, Z    +0.000, E1   +14.282, E3 +91609.488}
SPL {X  -162.808, Y  +378.562, Z    +0.000, E1    +4.298, E3 +91609.420}
SPL {X  -162.820, Y  +382.500, Z    +0.000, E1    +0.000, E3 +91608.993}
SPL {X  -162.820, Y  +384.915, Z    +0.000, E1    -4.894, E3 +91608.706}
SPL {X  -162.820, Y  +388.986, Z    +0.000, E1   -15.047, E3 +91608.804}
SPL {X  -162.820, Y  +393.007, Z    +0.000, E1   -25.093, E3 +91608.695}
SPL {X  -162.820, Y  +400.636, Z    +0.000, E1   -41.711, E3 +91608.745}
SPL {X  -162.820, Y  +414.705, Z    +0.000, E1   -61.052, E3 +91608.331}
SPL {X  -162.820, Y  +466.149, Z    +0.000, E1   -74.732, E3 +91618.327}
SPL {X  -160.722, Y  +699.554, Z    +0.000, E1   -75.485, E3 +91715.737}
SPL {X  -159.966, Y  +703.854, Z    +0.000, E1   -74.386, E3 +91730.641}
SPL {X  -156.868, Y  +717.123, Z    +0.000, E1   -74.182, E3 +91740.319}
SPL {X  -153.226, Y  +728.564, Z    +0.000, E1   -73.755, E3 +91751.327}
SPL {X  -149.090, Y  +738.941, Z    +0.000, E1   -73.348, E3 +91760.901}
SPL {X  -145.714, Y  +746.149, Z    +0.000, E1   -72.951, E3 +91768.487}
SPL {X  -140.946, Y  +755.015, Z    +0.000, E1   -72.452, E3 +91777.590}
SPL {X  -136.902, Y  +761.638, Z    +0.000, E1   -71.857, E3 +91785.457}
SPL {X  -133.350, Y  +766.925, Z    +0.000, E1   -71.498, E3 +91790.778}
SPL {X  -129.687, Y  +771.946, Z    +0.000, E1   -71.061, E3 +91796.144}
SPL {X  -126.374, Y  +776.164, Z    +0.000, E1   -70.494, E3 +91801.397}
SPL {X  -123.763, Y  +779.297, Z    +0.000, E1   -70.128, E3 +91804.773}
SPL {X  -119.350, Y  +784.252, Z    +0.000, E1   -71.016, E3 +91803.973}
SPL {X   -61.593, Y  +824.220, Z    +0.000, E1   -55.970, E3 +91970.289}
ENDSPLINE

SPLINE
SPL {X  -131.598, Y  +769.376, Z    +0.000, E1   -56.871, E3 +92136.560}
SPL {X  -152.760, Y  +729.846, Z    +0.000, E1   -44.713, E3 +92143.613}
SPL {X  -158.868, Y  +709.157, Z    +0.000, E1   -33.466, E3 +92144.814}
SPL {X  -161.987, Y  +689.949, Z    +0.000, E1   -18.777, E3 +92145.775}
SPL {X  -162.803, Y  +675.860, Z    +0.000, E1    -4.958, E3 +92145.757}
SPL {X  -162.820, Y  +671.500, Z    +0.000, E1    +0.000, E3 +92145.293}
SPL {X  -162.820, Y  +669.410, Z    +0.000, E1    +4.515, E3 +92145.056}
SPL {X  -162.820, Y  +664.781, Z    +0.000, E1   +16.411, E3 +92145.051}
SPL {X  -162.820, Y  +659.650, Z    +0.000, E1   +29.778, E3 +92145.061}
SPL {X  -162.820, Y  +654.031, Z    +0.000, E1   +42.449, E3 +92144.975}
SPL {X  -162.820, Y  +647.611, Z    +0.000, E1   +52.483, E3 +92145.505}
SPL {X  -162.820, Y  +637.134, Z    +0.000, E1   +65.232, E3 +92143.753}
SPL {X  -162.820, Y  +616.721, Z    +0.000, E1   +72.273, E3 +92147.487}
SPL {X  -162.820, Y  +577.172, Z    +0.000, E1   +75.843, E3 +92157.467}
SPL {X  -159.895, Y  +349.775, Z    +0.000, E1   +76.042, E3 +92249.133}
ENDSPLINE

SPLINE
SPL {X  -160.357, Y  +352.285, Z    +0.000, E1   +74.783, E3 +92262.071}
ENDSPLINE

SPLINE
SPL {X  -145.737, Y  +307.897, Z    +0.000, E1   +77.368, E3 +92254.646}
SPL {X  -145.122, Y  +306.676, Z    +0.000, E1   +76.360, E3 +92265.999}
ENDSPLINE

SPLINE
SPL {X  -145.186, Y  +306.802, Z    +0.000, E1   +74.850, E3 +92280.352}
ENDSPLINE

SPLINE
SPL {X  -143.742, Y  +304.025, Z    +0.000, E1   +73.644, E3 +92292.407}
SPL {X  -141.993, Y  +300.823, Z    +0.000, E1   +72.659, E3 +92301.979}
SPL {X  -138.166, Y  +294.358, Z    +0.000, E1   +72.281, E3 +92308.440}
SPL {X  -134.385, Y  +288.571, Z    +0.000, E1   +71.826, E3 +92314.704}
SPL {X  -129.872, Y  +282.297, Z    +0.000, E1   +71.229, E3 +92321.874}
SPL {X  -124.448, Y  +275.510, Z    +0.000, E1   +70.509, E3 +92329.247}
SPL {X  -117.513, Y  +267.801, Z    +0.000, E1   +72.197, E3 +92326.830}
SPL {X   -63.140, Y  +230.421, Z    +0.000, E1   +55.875, E3 +92496.268}
ENDSPLINE

SPLINE
SPL {X  -130.329, Y  +282.905, Z    +0.000, E1   +55.659, E3 +92654.604}
SPL {X  -150.766, Y  +319.018, Z    +0.000, E1   +45.408, E3 +92663.097}
SPL {X  -157.479, Y  +339.138, Z    +0.000, E1   +35.556, E3 +92664.532}
SPL {X  -160.994, Y  +356.185, Z    +0.000, E1   +24.373, E3 +92666.578}
SPL {X  -162.637, Y  +372.778, Z    +0.000, E1   +10.098, E3 +92666.598}
SPL {X  -162.820, Y  +382.419, Z    +0.000, E1    +0.163, E3 +92666.158}
SPL {X  -162.820, Y  +384.915, Z    +0.000, E1    -4.894, E3 +92665.849}
SPL {X  -162.820, Y  +388.986, Z    +0.000, E1   -15.047, E3 +92665.947}
SPL {X  -162.820, Y  +393.007, Z    +0.000, E1   -25.093, E3 +92665.838}
SPL {X  -162.820, Y  +400.636, Z    +0.000, E1   -41.711, E3 +92665.888}
SPL {X  -162.820, Y  +414.705, Z    +0.000, E1   -61.052, E3 +92665.474}
SPL {X  -162.820, Y  +466.149, Z    +0.000, E1   -74.732, E3 +92675.470}
SPL {X  -160.066, Y  +703.318, Z    +0.000, E1   -76.774, E3 +92760.318}
ENDSPLINE

SPLINE
SPL {X  -161.105, Y  +697.069, Z    +0.000, E1   -74.557, E3 +92781.932}
ENDSPLINE

SPLINE
SPL {X  -159.270, Y  +707.314, Z    +0.000, E1   -74.359, E3 +92789.956}
SPL {X  -156.868, Y  +717.123, Z    +0.000, E1   -74.182, E3 +92797.462}
SPL {X  -153.226, Y  +728.564, Z    +0.000, E1   -73.755, E3 +92808.470}
SPL {X  -149.090, Y  +738.941, Z    +0.000, E1   -73.348, E3 +92818.043}
SPL {X  -145.714, Y  +746.149, Z    +0.000, E1   -72.951, E3 +92825.630}
SPL {X  -140.946, Y  +755.015, Z    +0.000, E1   -72.452, E3 +92834.733}
SPL {X  -136.902, Y  +761.638, Z    +0.000, E1   -71.857, E3 +92842.600}
SPL {X  -133.350, Y  +766.925, Z    +0.000, E1   -71.498, E3 +92847.920}
SPL {X  -129.687, Y  +771.946, Z    +0.000, E1   -71.061, E3 +92853.286}
SPL {X  -126.374, Y  +776.164, Z    +0.000, E1   -70.494, E3 +92858.540}
SPL {X  -123.763, Y  +779.297, Z    +0.000, E1   -70.128, E3 +92861.916}
SPL {X  -119.350, Y  +784.252, Z    +0.000, E1   -71.016, E3 +92861.116}
SPL {X   -61.795, Y  +824.138, Z    +0.000, E1   -56.629, E3 +93007.263}
ENDSPLINE

SPLINE
SPL {X  -113.687, Y  +790.058, Z    +0.000, E1   -59.721, E3 +93184.010}
SPL {X  -139.151, Y  +758.042, Z    +0.000, E1   -54.091, E3 +93195.569}
SPL {X  -152.760, Y  +729.846, Z    +0.000, E1   -44.713, E3 +93200.756}
SPL {X  -158.868, Y  +709.157, Z    +0.000, E1   -33.466, E3 +93201.957}
SPL {X  -161.987, Y  +689.949, Z    +0.000, E1   -18.777, E3 +93202.918}
SPL {X  -162.743, Y  +678.515, Z    +0.000, E1    -7.658, E3 +93202.913}
SPL {X  -162.820, Y  +671.380, Z    +0.000, E1    +0.035, E3 +93202.418}
SPL {X  -162.820, Y  +668.318, Z    +0.000, E1    +7.404, E3 +93202.155}
SPL {X  -162.820, Y  +664.781, Z    +0.000, E1   +16.411, E3 +93202.194}
SPL {X  -162.820, Y  +659.650, Z    +0.000, E1   +29.778, E3 +93202.204}
SPL {X  -162.820, Y  +651.175, Z    +0.000, E1   +47.162, E3 +93202.353}
SPL {X  -162.820, Y  +633.243, Z    +0.000, E1   +67.111, E3 +93201.608}
SPL {X  -162.820, Y  +577.172, Z    +0.000, E1   +75.843, E3 +93214.610}
SPL {X  -159.895, Y  +349.775, Z    +0.000, E1   +76.042, E3 +93306.276}
ENDSPLINE

SPLINE
SPL {X  -160.357, Y  +352.285, Z    +0.000, E1   +74.783, E3 +93319.214}
ENDSPLINE

SPLINE
SPL {X  -145.737, Y  +307.897, Z    +0.000, E1   +77.368, E3 +93311.789}
SPL {X  -145.122, Y  +306.676, Z    +0.000, E1   +76.360, E3 +93323.142}
ENDSPLINE

SPLINE
SPL {X  -145.186, Y  +306.802, Z    +0.000, E1   +74.850, E3 +93337.495}
ENDSPLINE

SPLINE
SPL {X  -143.742, Y  +304.025, Z    +0.000, E1   +73.644, E3 +93349.550}
SPL {X  -141.993, Y  +300.823, Z    +0.000, E1   +72.659, E3 +93359.122}
SPL {X  -138.166, Y  +294.358, Z    +0.000, E1   +72.281, E3 +93365.583}
SPL {X  -134.385, Y  +288.571, Z    +0.000, E1   +71.826, E3 +93371.847}
SPL {X  -130.773, Y  +283.501, Z    +0.000, E1   +71.398, E3 +93377.271}
SPL {X  -126.922, Y  +278.513, Z    +0.000, E1   +70.767, E3 +93383.425}
SPL {X  -123.520, Y  +274.419, Z    +0.000, E1   +70.342, E3 +93387.624}
SPL {X  -117.513, Y  +267.801, Z    +0.000, E1   +72.197, E3 +93383.972}
SPL {X   -63.140, Y  +230.421, Z    +0.000, E1   +55.875, E3 +93553.411}
ENDSPLINE

SPLINE
SPL {X  -130.329, Y  +282.905, Z    +0.000, E1   +55.659, E3 +93711.747}
SPL {X  -150.766, Y  +319.018, Z    +0.000, E1   +45.408, E3 +93720.240}
SPL {X  -157.479, Y  +339.138, Z    +0.000, E1   +35.556, E3 +93721.675}
SPL {X  -160.994, Y  +356.185, Z    +0.000, E1   +24.373, E3 +93723.721}
SPL {X  -162.352, Y  +368.168, Z    +0.000, E1   +14.282, E3 +93723.774}
SPL {X  -162.808, Y  +378.562, Z    +0.000, E1    +4.298, E3 +93723.706}
SPL {X  -162.820, Y  +382.500, Z    +0.000, E1    +0.000, E3 +93723.278}
SPL {X  -162.820, Y  +384.915, Z    +0.000, E1    -4.894, E3 +93722.992}
SPL {X  -162.820, Y  +388.986, Z    +0.000, E1   -15.047, E3 +93723.090}
SPL {X  -162.820, Y  +394.732, Z    +0.000, E1   -28.992, E3 +93722.941}
SPL {X  -162.820, Y  +403.075, Z    +0.000, E1   -46.096, E3 +93723.171}
SPL {X  -162.820, Y  +414.705, Z    +0.000, E1   -61.052, E3 +93722.617}
SPL {X  -162.820, Y  +466.149, Z    +0.000, E1   -74.732, E3 +93732.613}
SPL {X  -160.722, Y  +699.554, Z    +0.000, E1   -75.485, E3 +93830.023}
SPL {X  -159.966, Y  +703.854, Z    +0.000, E1   -74.386, E3 +93844.926}
SPL {X  -156.868, Y  +717.123, Z    +0.000, E1   -74.182, E3 +93854.605}
SPL {X  -153.226, Y  +728.564, Z    +0.000, E1   -73.755, E3 +93865.613}
SPL {X  -149.090, Y  +738.941, Z    +0.000, E1   -73.348, E3 +93875.186}
SPL {X  -145.714, Y  +746.149, Z    +0.000, E1   -72.951, E3 +93882.773}
SPL {X  -140.946, Y  +755.015, Z    +0.000, E1   -72.452, E3 +93891.876}
SPL {X  -136.902, Y  +761.638, Z    +0.000, E1   -71.857, E3 +93899.743}
SPL {X  -133.350, Y  +766.925, Z    +0.000, E1   -71.498, E3 +93905.063}
SPL {X  -129.687, Y  +771.946, Z    +0.000, E1   -71.061, E3 +93910.429}
SPL {X  -126.374, Y  +776.164, Z    +0.000, E1   -70.494, E3 +93915.683}
SPL {X  -122.717, Y  +780.508, Z    +0.000, E1   -70.361, E3 +93918.720}
SPL {X  -114.093, Y  +789.660, Z    +0.000, E1   -71.634, E3 +93918.738}
SPL {X   -61.593, Y  +824.220, Z    +0.000, E1   -55.970, E3 +94084.574}
ENDSPLINE

SPLINE
SPL {X  -131.598, Y  +769.376, Z    +0.000, E1   -56.871, E3 +94250.846}
SPL {X  -152.760, Y  +729.846, Z    +0.000, E1   -44.713, E3 +94257.898}
SPL {X  -158.868, Y  +709.157, Z    +0.000, E1   -33.466, E3 +94259.099}
SPL {X  -161.987, Y  +689.949, Z    +0.000, E1   -18.777, E3 +94260.061}
SPL {X  -162.743, Y  +678.515, Z    +0.000, E1    -7.658, E3 +94260.056}
SPL {X  -162.820, Y  +671.380, Z    +0.000, E1    +0.035, E3 +94259.560}
SPL {X  -162.820, Y  +668.318, Z    +0.000, E1    +7.404, E3 +94259.298}
SPL {X  -162.820, Y  +664.781, Z    +0.000, E1   +16.411, E3 +94259.337}
SPL {X  -162.820, Y  +659.650, Z    +0.000, E1   +29.778, E3 +94259.346}
SPL {X  -162.820, Y  +654.031, Z    +0.000, E1   +42.449, E3 +94259.260}
SPL {X  -162.820, Y  +647.611, Z    +0.000, E1   +52.483, E3 +94259.791}
SPL {X  -162.820, Y  +637.134, Z    +0.000, E1   +65.232, E3 +94258.039}
SPL {X  -162.820, Y  +616.721, Z    +0.000, E1   +72.273, E3 +94261.773}
SPL {X  -162.820, Y  +577.172, Z    +0.000, E1   +75.843, E3 +94271.753}
SPL {X  -159.895, Y  +349.775, Z    +0.000, E1   +76.042, E3 +94363.419}
ENDSPLINE

SPLINE
SPL {X  -160.357, Y  +352.285, Z    +0.000, E1   +74.783, E3 +94376.357}
ENDSPLINE

SPLINE
SPL {X  -145.737, Y  +307.897, Z    +0.000, E1   +77.368, E3 +94368.932}
SPL {X  -145.329, Y  +307.084, Z    +0.000, E1   +76.571, E3 +94377.768}
ENDSPLINE

SPLINE
SPL {X  -145.355, Y  +307.136, Z    +0.000, E1   +75.607, E3 +94387.292}
ENDSPLINE

SPLINE
SPL {X  -144.515, Y  +305.495, Z    +0.000, E1   +74.543, E3 +94398.101}
SPL {X  -143.690, Y  +303.925, Z    +0.000, E1   +73.372, E3 +94408.840}
SPL {X  -141.993, Y  +300.823, Z    +0.000, E1   +72.659, E3 +94416.265}
SPL {X  -138.166, Y  +294.358, Z    +0.000, E1   +72.281, E3 +94422.726}
SPL {X  -134.385, Y  +288.571, Z    +0.000, E1   +71.826, E3 +94428.990}
SPL {X  -130.773, Y  +283.501, Z    +0.000, E1   +71.398, E3 +94434.414}
SPL {X  -126.922, Y  +278.513, Z    +0.000, E1   +70.767, E3 +94440.568}
SPL {X  -123.520, Y  +274.419, Z    +0.000, E1   +70.342, E3 +94444.767}
SPL {X  -117.513, Y  +267.801, Z    +0.000, E1   +72.197, E3 +94441.115}
SPL {X   -63.140, Y  +230.421, Z    +0.000, E1   +55.875, E3 +94610.554}
ENDSPLINE

SPLINE
SPL {X  -130.329, Y  +282.905, Z    +0.000, E1   +55.659, E3 +94768.890}
SPL {X  -154.728, Y  +329.807, Z    +0.000, E1   +40.640, E3 +94778.271}
SPL {X  -160.994, Y  +356.185, Z    +0.000, E1   +24.373, E3 +94780.864}
SPL {X  -162.637, Y  +372.778, Z    +0.000, E1   +10.098, E3 +94780.884}
SPL {X  -162.820, Y  +382.748, Z    +0.000, E1    -0.178, E3 +94780.377}
SPL {X  -162.820, Y  +387.647, Z    +0.000, E1   -11.488, E3 +94780.166}
SPL {X  -162.820, Y  +393.007, Z    +0.000, E1   -25.093, E3 +94780.124}
SPL {X  -162.820, Y  +400.636, Z    +0.000, E1   -41.711, E3 +94780.173}
SPL {X  -162.820, Y  +414.705, Z    +0.000, E1   -61.052, E3 +94779.760}
SPL {X  -162.820, Y  +466.149, Z    +0.000, E1   -74.732, E3 +94789.756}
SPL {X  -160.066, Y  +703.318, Z    +0.000, E1   -76.774, E3 +94874.603}
ENDSPLINE

SPLINE
SPL {X  -161.105, Y  +697.069, Z    +0.000, E1   -74.557, E3 +94896.218}
ENDSPLINE

SPLINE
SPL {X  -159.270, Y  +707.314, Z    +0.000, E1   -74.359, E3 +94904.241}
SPL {X  -156.868, Y  +717.123, Z    +0.000, E1   -74.182, E3 +94911.747}
SPL {X  -153.226, Y  +728.564, Z    +0.000, E1   -73.755, E3 +94922.756}
SPL {X  -149.090, Y  +738.941, Z    +0.000, E1   -73.348, E3 +94932.329}
SPL {X  -145.714, Y  +746.149, Z    +0.000, E1   -72.951, E3 +94939.916}
SPL {X  -142.592, Y  +752.100, Z    +0.000, E1   -72.554, E3 +94946.449}
SPL {X  -139.608, Y  +757.285, Z    +0.000, E1   -72.326, E3 +94951.118}
SPL {X  -136.902, Y  +761.638, Z    +0.000, E1   -71.857, E3 +94956.886}
SPL {X  -133.350, Y  +766.925, Z    +0.000, E1   -71.498, E3 +94962.206}
SPL {X  -129.687, Y  +771.946, Z    +0.000, E1   -71.061, E3 +94967.572}
SPL {X  -126.374, Y  +776.164, Z    +0.000, E1   -70.494, E3 +94972.826}
SPL {X  -123.763, Y  +779.297, Z    +0.000, E1   -70.128, E3 +94976.201}
SPL {X  -119.350, Y  +784.252, Z    +0.000, E1   -71.016, E3 +94975.402}
SPL {X   -61.795, Y  +824.138, Z    +0.000, E1   -56.629, E3 +95121.549}
ENDSPLINE

SPLINE
SPL {X  -113.687, Y  +790.058, Z    +0.000, E1   -59.721, E3 +95298.296}
SPL {X  -139.151, Y  +758.042, Z    +0.000, E1   -54.091, E3 +95309.855}
SPL {X  -152.760, Y  +729.846, Z    +0.000, E1   -44.713, E3 +95315.041}
SPL {X  -158.868, Y  +709.157, Z    +0.000, E1   -33.466, E3 +95316.242}
SPL {X  -161.987, Y  +689.949, Z    +0.000, E1   -18.777, E3 +95317.203}
SPL {X  -162.743, Y  +678.515, Z    +0.000, E1    -7.658, E3 +95317.199}
SPL {X  -162.820, Y  +671.380, Z    +0.000, E1    +0.035, E3 +95316.703}
SPL {X  -162.820, Y  +668.318, Z    +0.000, E1    +7.404, E3 +95316.440}
SPL {X  -162.820, Y  +664.781, Z    +0.000, E1   +16.411, E3 +95316.480}
SPL {X  -162.820, Y  +659.650, Z    +0.000, E1   +29.778, E3 +95316.489}
SPL {X  -162.820, Y  +654.031, Z    +0.000, E1   +42.449, E3 +95316.403}
SPL {X  -162.820, Y  +647.611, Z    +0.000, E1   +52.483, E3 +95316.933}
SPL {X  -162.820, Y  +637.134, Z    +0.000, E1   +65.232, E3 +95315.181}
SPL {X  -162.820, Y  +616.721, Z    +0.000, E1   +72.273, E3 +95318.915}
SPL {X  -162.820, Y  +577.172, Z    +0.000, E1   +75.843, E3 +95328.896}
SPL {X  -159.895, Y  +349.775, Z    +0.000, E1   +76.042, E3 +95420.562}
ENDSPLINE

SPLINE
SPL {X  -160.357, Y  +352.285, Z    +0.000, E1   +74.783, E3 +95433.500}
ENDSPLINE

SPLINE
SPL {X  -145.737, Y  +307.897, Z    +0.000, E1   +77.368, E3 +95426.075}
SPL {X  -145.329, Y  +307.084, Z    +0.000, E1   +76.571, E3 +95434.911}
ENDSPLINE

SPLINE
SPL {X  -145.355, Y  +307.136, Z    +0.000, E1   +75.607, E3 +95444.435}
ENDSPLINE

SPLINE
SPL {X  -144.515, Y  +305.495, Z    +0.000, E1   +74.543, E3 +95455.244}
SPL {X  -143.690, Y  +303.925, Z    +0.000, E1   +73.372, E3 +95465.983}
SPL {X  -141.993, Y  +300.823, Z    +0.000, E1   +72.659, E3 +95473.408}
SPL {X  -138.166, Y  +294.358, Z    +0.000, E1   +72.281, E3 +95479.869}
SPL {X  -134.385, Y  +288.571, Z    +0.000, E1   +71.826, E3 +95486.132}
SPL {X  -129.872, Y  +282.297, Z    +0.000, E1   +71.229, E3 +95493.303}
SPL {X  -124.448, Y  +275.510, Z    +0.000, E1   +70.509, E3 +95500.675}
SPL {X  -117.513, Y  +267.801, Z    +0.000, E1   +72.197, E3 +95498.258}
SPL {X   -63.140, Y  +230.421, Z    +0.000, E1   +55.875, E3 +95667.697}
ENDSPLINE

SPLINE
SPL {X  -130.329, Y  +282.905, Z    +0.000, E1   +55.659, E3 +95826.033}
SPL {X  -150.766, Y  +319.018, Z    +0.000, E1   +45.408, E3 +95834.525}
SPL {X  -157.479, Y  +339.138, Z    +0.000, E1   +35.556, E3 +95835.961}
SPL {X  -160.994, Y  +356.185, Z    +0.000, E1   +24.373, E3 +95838.007}
SPL {X  -162.637, Y  +372.778, Z    +0.000, E1   +10.098, E3 +95838.027}
SPL {X  -162.820, Y  +382.748, Z    +0.000, E1    -0.178, E3 +95837.520}
SPL {X  -162.820, Y  +387.647, Z    +0.000, E1   -11.488, E3 +95837.308}
SPL {X  -162.820, Y  +393.007, Z    +0.000, E1   -25.093, E3 +95837.266}
SPL {X  -162.820, Y  +400.636, Z    +0.000, E1   -41.711, E3 +95837.316}
SPL {X  -162.820, Y  +414.705, Z    +0.000, E1   -61.052, E3 +95836.903}
SPL {X  -162.820, Y  +466.149, Z    +0.000, E1   -74.732, E3 +95846.899}
SPL {X  -160.722, Y  +699.554, Z    +0.000, E1   -75.485, E3 +95944.309}
SPL {X  -159.966, Y  +703.854, Z    +0.000, E1   -74.386, E3 +95959.212}
SPL {X  -156.868, Y  +717.123, Z    +0.000, E1   -74.182, E3 +95968.890}
SPL {X  -154.373, Y  +725.261, Z    +0.000, E1   -73.879, E3 +95976.600}
SPL {X  -152.060, Y  +731.708, Z    +0.000, E1   -73.572, E3 +95983.248}
SPL {X  -149.090, Y  +738.941, Z    +0.000, E1   -73.348, E3 +95989.472}
SPL {X  -145.714, Y  +746.149, Z    +0.000, E1   -72.951, E3 +95997.059}
SPL {X  -140.946, Y  +755.015, Z    +0.000, E1   -72.452, E3 +96006.162}
SPL {X  -136.902, Y  +761.638, Z    +0.000, E1   -71.857, E3 +96014.028}
SPL {X  -133.350, Y  +766.925, Z    +0.000, E1   -71.498, E3 +96019.349}
SPL {X  -129.687, Y  +771.946, Z    +0.000, E1   -71.061, E3 +96024.715}
SPL {X  -126.374, Y  +776.164, Z    +0.000, E1   -70.494, E3 +96029.968}
SPL {X  -123.763, Y  +779.297, Z    +0.000, E1   -70.128, E3 +96033.344}
SPL {X  -119.350, Y  +784.252, Z    +0.000, E1   -71.016, E3 +96032.544}
SPL {X   -61.795, Y  +824.138, Z    +0.000, E1   -56.629, E3 +96178.692}
ENDSPLINE

SPLINE
SPL {X  -113.687, Y  +790.058, Z    +0.000, E1   -59.721, E3 +96355.439}
SPL {X  -139.151, Y  +758.042, Z    +0.000, E1   -54.091, E3 +96366.998}
SPL {X  -152.760, Y  +729.846, Z    +0.000, E1   -44.713, E3 +96372.184}
SPL {X  -158.868, Y  +709.157, Z    +0.000, E1   -33.466, E3 +96373.385}
SPL {X  -161.987, Y  +689.949, Z    +0.000, E1   -18.777, E3 +96374.346}
SPL {X  -162.743, Y  +678.515, Z    +0.000, E1    -7.658, E3 +96374.342}
SPL {X  -162.820, Y  +671.380, Z    +0.000, E1    +0.035, E3 +96373.846}
SPL {X  -162.820, Y  +668.318, Z    +0.000, E1    +7.404, E3 +96373.583}
SPL {X  -162.820, Y  +664.781, Z    +0.000, E1   +16.411, E3 +96373.622}
SPL {X  -162.820, Y  +659.650, Z    +0.000, E1   +29.778, E3 +96373.632}
SPL {X  -162.820, Y  +651.175, Z    +0.000, E1   +47.162, E3 +96373.782}
SPL {X  -162.820, Y  +633.243, Z    +0.000, E1   +67.111, E3 +96373.037}
SPL {X  -162.820, Y  +577.172, Z    +0.000, E1   +75.843, E3 +96386.039}
SPL {X  -159.895, Y  +349.775, Z    +0.000, E1   +76.042, E3 +96477.705}
ENDSPLINE

SPLINE
SPL {X  -160.357, Y  +352.285, Z    +0.000, E1   +74.783, E3 +96490.642}
ENDSPLINE

SPLINE
SPL {X  -145.737, Y  +307.897, Z    +0.000, E1   +77.368, E3 +96483.218}
SPL {X  -145.122, Y  +306.676, Z    +0.000, E1   +76.360, E3 +96494.571}
ENDSPLINE

SPLINE
SPL {X  -145.186, Y  +306.802, Z    +0.000, E1   +74.850, E3 +96508.924}
ENDSPLINE

SPLINE
SPL {X  -143.742, Y  +304.025, Z    +0.000, E1   +73.644, E3 +96520.978}
SPL {X  -141.993, Y  +300.823, Z    +0.000, E1   +72.659, E3 +96530.551}
SPL {X  -138.166, Y  +294.358, Z    +0.000, E1   +72.281, E3 +96537.012}
SPL {X  -134.385, Y  +288.571, Z    +0.000, E1   +71.826, E3 +96543.275}
SPL {X  -130.773, Y  +283.501, Z    +0.000, E1   +71.398, E3 +96548.700}
SPL {X  -126.922, Y  +278.513, Z    +0.000, E1   +70.767, E3 +96554.854}
SPL {X  -123.520, Y  +274.419, Z    +0.000, E1   +70.342, E3 +96559.052}
SPL {X  -117.513, Y  +267.801, Z    +0.000, E1   +72.197, E3 +96555.401}
SPL {X   -63.140, Y  +230.421, Z    +0.000, E1   +55.875, E3 +96724.840}
ENDSPLINE

SPLINE
SPL {X  -130.329, Y  +282.905, Z    +0.000, E1   +55.659, E3 +96883.176}
SPL {X  -154.728, Y  +329.807, Z    +0.000, E1   +40.640, E3 +96892.557}
SPL {X  -160.994, Y  +356.185, Z    +0.000, E1   +24.373, E3 +96895.150}
SPL {X  -162.637, Y  +372.778, Z    +0.000, E1   +10.098, E3 +96895.170}
SPL {X  -162.820, Y  +382.748, Z    +0.000, E1    -0.178, E3 +96894.662}
SPL {X  -162.820, Y  +387.647, Z    +0.000, E1   -11.488, E3 +96894.451}
SPL {X  -162.820, Y  +393.007, Z    +0.000, E1   -25.093, E3 +96894.409}
SPL {X  -162.820, Y  +400.636, Z    +0.000, E1   -41.711, E3 +96894.459}
SPL {X  -162.820, Y  +414.705, Z    +0.000, E1   -61.052, E3 +96894.046}
SPL {X  -162.820, Y  +466.149, Z    +0.000, E1   -74.732, E3 +96904.042}
SPL {X  -160.722, Y  +699.554, Z    +0.000, E1   -75.485, E3 +97001.452}
SPL {X  -159.966, Y  +703.854, Z    +0.000, E1   -74.386, E3 +97016.355}
SPL {X  -156.868, Y  +717.123, Z    +0.000, E1   -74.182, E3 +97026.033}
SPL {X  -154.373, Y  +725.261, Z    +0.000, E1   -73.879, E3 +97033.743}
SPL {X  -152.060, Y  +731.708, Z    +0.000, E1   -73.572, E3 +97040.391}
SPL {X  -149.090, Y  +738.941, Z    +0.000, E1   -73.348, E3 +97046.615}
SPL {X  -145.714, Y  +746.149, Z    +0.000, E1   -72.951, E3 +97054.202}
SPL {X  -140.946, Y  +755.015, Z    +0.000, E1   -72.452, E3 +97063.305}
SPL {X  -136.902, Y  +761.638, Z    +0.000, E1   -71.857, E3 +97071.171}
SPL {X  -133.350, Y  +766.925, Z    +0.000, E1   -71.498, E3 +97076.492}
SPL {X  -129.687, Y  +771.946, Z    +0.000, E1   -71.061, E3 +97081.858}
SPL {X  -126.374, Y  +776.164, Z    +0.000, E1   -70.494, E3 +97087.111}
SPL {X  -123.763, Y  +779.297, Z    +0.000, E1   -70.128, E3 +97090.487}
SPL {X  -119.350, Y  +784.252, Z    +0.000, E1   -71.016, E3 +97089.687}
SPL {X   -61.795, Y  +824.138, Z    +0.000, E1   -56.629, E3 +97235.834}
ENDSPLINE

SPLINE
SPL {X  -113.687, Y  +790.058, Z    +0.000, E1   -59.721, E3 +97412.582}
SPL {X  -139.151, Y  +758.042, Z    +0.000, E1   -54.091, E3 +97424.141}
SPL {X  -152.760, Y  +729.846, Z    +0.000, E1   -44.713, E3 +97429.327}
SPL {X  -158.868, Y  +709.157, Z    +0.000, E1   -33.466, E3 +97430.528}
SPL {X  -161.987, Y  +689.949, Z    +0.000, E1   -18.777, E3 +97431.489}
SPL {X  -162.803, Y  +675.860, Z    +0.000, E1    -4.958, E3 +97431.471}
SPL {X  -162.820, Y  +671.500, Z    +0.000, E1    +0.000, E3 +97431.008}
SPL {X  -162.820, Y  +669.410, Z    +0.000, E1    +4.515, E3 +97430.770}
SPL {X  -162.820, Y  +664.781, Z    +0.000, E1   +16.411, E3 +97430.765}
SPL {X  -162.820, Y  +659.650, Z    +0.000, E1   +29.778, E3 +97430.775}
SPL {X  -162.820, Y  +651.175, Z    +0.000, E1   +47.162, E3 +97430.925}
SPL {X  -162.820, Y  +637.134, Z    +0.000, E1   +65.232, E3 +97429.467}
SPL {X  -162.820, Y  +616.721, Z    +0.000, E1   +72.273, E3 +97433.201}
SPL {X  -162.820, Y  +577.172, Z    +0.000, E1   +75.843, E3 +97443.181}
SPL {X  -159.895, Y  +349.775, Z    +0.000, E1   +76.042, E3 +97534.848}
ENDSPLINE

SPLINE
SPL {X  -160.357, Y  +352.285, Z    +0.000, E1   +74.783, E3 +97547.785}
ENDSPLINE

SPLINE
SPL {X  -145.737, Y  +307.897, Z    +0.000, E1   +77.368, E3 +97540.361}
SPL {X  -145.329, Y  +307.084, Z    +0.000, E1   +76.571, E3 +97549.197}
ENDSPLINE

SPLINE
SPL {X  -145.355, Y  +307.136, Z    +0.000, E1   +75.607, E3 +97558.721}
ENDSPLINE

SPLINE
SPL {X  -144.515, Y  +305.495, Z    +0.000, E1   +74.543, E3 +97569.530}
SPL {X  -143.690, Y  +303.925, Z    +0.000, E1   +73.372, E3 +97580.269}
SPL {X  -141.993, Y  +300.823, Z    +0.000, E1   +72.659, E3 +97587.693}
SPL {X  -138.166, Y  +294.358, Z    +0.000, E1   +72.281, E3 +97594.155}
SPL {X  -134.385, Y  +288.571, Z    +0.000, E1   +71.826, E3 +97600.418}
SPL {X  -130.773, Y  +283.501, Z    +0.000, E1   +71.398, E3 +97605.842}
SPL {X  -126.922, Y  +278.513, Z    +0.000, E1   +70.767, E3 +97611.996}
SPL {X  -123.520, Y  +274.419, Z    +0.000, E1   +70.342, E3 +97616.195}
SPL {X  -117.513, Y  +267.801, Z    +0.000, E1   +72.197, E3 +97612.544}
SPL {X   -63.140, Y  +230.421, Z    +0.000, E1   +55.875, E3 +97781.983}
ENDSPLINE

SPLINE
SPL {X  -130.329, Y  +282.905, Z    +0.000, E1   +55.659, E3 +97940.318}
SPL {X  -154.728, Y  +329.807, Z    +0.000, E1   +40.640, E3 +97949.700}
SPL {X  -160.994, Y  +356.185, Z    +0.000, E1   +24.373, E3 +97952.293}
SPL {X  -162.637, Y  +372.778, Z    +0.000, E1   +10.098, E3 +97952.313}
SPL {X  -162.820, Y  +382.748, Z    +0.000, E1    -0.178, E3 +97951.805}
SPL {X  -162.820, Y  +387.647, Z    +0.000, E1   -11.488, E3 +97951.594}
SPL {X  -162.820, Y  +393.007, Z    +0.000, E1   -25.093, E3 +97951.552}
SPL {X  -162.820, Y  +400.636, Z    +0.000, E1   -41.711, E3 +97951.602}
SPL {X  -162.820, Y  +414.705, Z    +0.000, E1   -61.052, E3 +97951.188}
SPL {X  -162.820, Y  +466.149, Z    +0.000, E1   -74.732, E3 +97961.185}
SPL {X  -160.066, Y  +703.318, Z    +0.000, E1   -76.774, E3 +98046.032}
ENDSPLINE

SPLINE
SPL {X  -161.105, Y  +697.069, Z    +0.000, E1   -74.557, E3 +98067.646}
ENDSPLINE

SPLINE
SPL {X  -159.270, Y  +707.314, Z    +0.000, E1   -74.359, E3 +98075.670}
SPL {X  -156.868, Y  +717.123, Z    +0.000, E1   -74.182, E3 +98083.176}
SPL {X  -153.226, Y  +728.564, Z    +0.000, E1   -73.755, E3 +98094.184}
SPL {X  -149.090, Y  +738.941, Z    +0.000, E1   -73.348, E3 +98103.758}
SPL {X  -145.714, Y  +746.149, Z    +0.000, E1   -72.951, E3 +98111.345}
SPL {X  -142.592, Y  +752.100, Z    +0.000, E1   -72.554, E3 +98117.877}
SPL {X  -139.608, Y  +757.285, Z    +0.000, E1   -72.326, E3 +98122.547}
SPL {X  -136.902, Y  +761.638, Z    +0.000, E1   -71.857, E3 +98128.314}
SPL {X  -133.350, Y  +766.925, Z    +0.000, E1   -71.498, E3 +98133.635}
SPL {X  -129.687, Y  +771.946, Z    +0.000, E1   -71.061, E3 +98139.001}
SPL {X  -126.374, Y  +776.164, Z    +0.000, E1   -70.494, E3 +98144.254}
SPL {X  -123.763, Y  +779.297, Z    +0.000, E1   -70.128, E3 +98147.630}
SPL {X  -119.350, Y  +784.252, Z    +0.000, E1   -71.016, E3 +98146.830}
SPL {X   -61.795, Y  +824.138, Z    +0.000, E1   -56.629, E3 +98292.977}
ENDSPLINE

SPLINE
SPL {X  -113.687, Y  +790.058, Z    +0.000, E1   -59.721, E3 +98469.724}
SPL {X  -139.151, Y  +758.042, Z    +0.000, E1   -54.091, E3 +98481.284}
SPL {X  -152.760, Y  +729.846, Z    +0.000, E1   -44.713, E3 +98486.470}
SPL {X  -158.868, Y  +709.157, Z    +0.000, E1   -33.466, E3 +98487.671}
SPL {X  -161.987, Y  +689.949, Z    +0.000, E1   -18.777, E3 +98488.632}
SPL {X  -162.803, Y  +675.860, Z    +0.000, E1    -4.958, E3 +98488.614}
SPL {X  -162.820, Y  +671.500, Z    +0.000, E1    +0.000, E3 +98488.151}
SPL {X  -162.820, Y  +669.410, Z    +0.000, E1    +4.515, E3 +98487.913}
SPL {X  -162.820, Y  +664.781, Z    +0.000, E1   +16.411, E3 +98487.908}
SPL {X  -162.820, Y  +659.650, Z    +0.000, E1   +29.778, E3 +98487.918}
SPL {X  -162.820, Y  +651.175, Z    +0.000, E1   +47.162, E3 +98488.068}
SPL {X  -162.820, Y  +633.243, Z    +0.000, E1   +67.111, E3 +98487.323}
SPL {X  -162.820, Y  +577.172, Z    +0.000, E1   +75.843, E3 +98500.324}
SPL {X  -159.895, Y  +349.775, Z    +0.000, E1   +76.042, E3 +98591.990}
ENDSPLINE

SPLINE
SPL {X  -160.357, Y  +352.285, Z    +0.000, E1   +74.783, E3 +98604.928}
ENDSPLINE

SPLINE
SPL {X  -145.737, Y  +307.897, Z    +0.000, E1   +77.368, E3 +98597.503}
SPL {X  -145.329, Y  +307.084, Z    +0.000, E1   +76.571, E3 +98606.340}
ENDSPLINE

SPLINE
SPL {X  -145.355, Y  +307.136, Z    +0.000, E1   +75.607, E3 +98615.864}
ENDSPLINE

SPLINE
SPL {X  -144.515, Y  +305.495, Z    +0.000, E1   +74.543, E3 +98626.673}
SPL {X  -143.690, Y  +303.925, Z    +0.000, E1   +73.372, E3 +98637.412}
SPL {X  -141.993, Y  +300.823, Z    +0.000, E1   +72.659, E3 +98644.836}
SPL {X  -138.166, Y  +294.358, Z    +0.000, E1   +72.281, E3 +98651.297}
SPL {X  -134.385, Y  +288.571, Z    +0.000, E1   +71.826, E3 +98657.561}
SPL {X  -130.773, Y  +283.501, Z    +0.000, E1   +71.398, E3 +98662.985}
SPL {X  -126.922, Y  +278.513, Z    +0.000, E1   +70.767, E3 +98669.139}
SPL {X  -123.520, Y  +274.419, Z    +0.000, E1   +70.342, E3 +98673.338}
SPL {X  -117.513, Y  +267.801, Z    +0.000, E1   +72.197, E3 +98669.687}
SPL {X   -63.140, Y  +230.421, Z    +0.000, E1   +55.875, E3 +98839.125}
ENDSPLINE

SPLINE
SPL {X  -130.329, Y  +282.905, Z    +0.000, E1   +55.659, E3 +98997.461}
SPL {X  -150.766, Y  +319.018, Z    +0.000, E1   +45.408, E3 +99005.954}
SPL {X  -157.479, Y  +339.138, Z    +0.000, E1   +35.556, E3 +99007.390}
SPL {X  -160.994, Y  +356.185, Z    +0.000, E1   +24.373, E3 +99009.435}
SPL {X  -162.352, Y  +368.168, Z    +0.000, E1   +14.282, E3 +99009.488}
SPL {X  -162.808, Y  +378.562, Z    +0.000, E1    +4.298, E3 +99009.420}
SPL {X  -162.820, Y  +382.500, Z    +0.000, E1    +0.000, E3 +99008.993}
SPL {X  -162.820, Y  +383.794, Z    +0.000, E1    -2.626, E3 +99008.734}
SPL {X  -162.820, Y  +387.647, Z    +0.000, E1   -11.488, E3 +99008.737}
SPL {X  -162.820, Y  +393.007, Z    +0.000, E1   -25.093, E3 +99008.695}
SPL {X  -162.820, Y  +400.636, Z    +0.000, E1   -41.711, E3 +99008.745}
SPL {X  -162.820, Y  +414.705, Z    +0.000, E1   -61.052, E3 +99008.331}
SPL {X  -162.820, Y  +466.149, Z    +0.000, E1   -74.732, E3 +99018.327}
SPL {X  -160.066, Y  +703.318, Z    +0.000, E1   -76.774, E3 +99103.175}
ENDSPLINE

SPLINE
SPL {X  -161.105, Y  +697.069, Z    +0.000, E1   -74.557, E3 +99124.789}
ENDSPLINE

SPLINE
SPL {X  -159.270, Y  +707.314, Z    +0.000, E1   -74.359, E3 +99132.813}
SPL {X  -156.868, Y  +717.123, Z    +0.000, E1   -74.182, E3 +99140.319}
SPL {X  -153.226, Y  +728.564, Z    +0.000, E1   -73.755, E3 +99151.327}
SPL {X  -149.090, Y  +738.941, Z    +0.000, E1   -73.348, E3 +99160.901}
SPL {X  -145.714, Y  +746.149, Z    +0.000, E1   -72.951, E3 +99168.487}
SPL {X  -140.946, Y  +755.015, Z    +0.000, E1   -72.452, E3 +99177.590}
SPL {X  -136.902, Y  +761.638, Z    +0.000, E1   -71.857, E3 +99185.457}
SPL {X  -133.350, Y  +766.925, Z    +0.000, E1   -71.498, E3 +99190.778}
SPL {X  -129.687, Y  +771.946, Z    +0.000, E1   -71.061, E3 +99196.144}
SPL {X  -126.374, Y  +776.164, Z    +0.000, E1   -70.494, E3 +99201.397}
SPL {X  -123.763, Y  +779.297, Z    +0.000, E1   -70.128, E3 +99204.773}
SPL {X  -119.350, Y  +784.252, Z    +0.000, E1   -71.016, E3 +99203.973}
SPL {X   -61.593, Y  +824.220, Z    +0.000, E1   -55.970, E3 +99370.289}
ENDSPLINE

SPLINE
SPL {X  -131.598, Y  +769.376, Z    +0.000, E1   -56.871, E3 +99536.560}
SPL {X  -152.760, Y  +729.846, Z    +0.000, E1   -44.713, E3 +99543.613}
SPL {X  -158.868, Y  +709.157, Z    +0.000, E1   -33.466, E3 +99544.814}
SPL {X  -161.987, Y  +689.949, Z    +0.000, E1   -18.777, E3 +99545.775}
SPL {X  -162.743, Y  +678.515, Z    +0.000, E1    -7.658, E3 +99545.770}
SPL {X  -162.820, Y  +671.588, Z    +0.000, E1    -0.190, E3 +99545.316}
SPL {X  -162.820, Y  +669.410, Z    +0.000, E1    +4.515, E3 +99545.056}
SPL {X  -162.820, Y  +664.781, Z    +0.000, E1   +16.411, E3 +99545.051}
SPL {X  -162.820, Y  +659.650, Z    +0.000, E1   +29.778, E3 +99545.061}
SPL {X  -162.820, Y  +654.031, Z    +0.000, E1   +42.449, E3 +99544.975}
SPL {X  -162.820, Y  +647.611, Z    +0.000, E1   +52.483, E3 +99545.505}
SPL {X  -162.820, Y  +637.134, Z    +0.000, E1   +65.232, E3 +99543.753}
SPL {X  -162.820, Y  +616.721, Z    +0.000, E1   +72.273, E3 +99547.487}
SPL {X  -162.820, Y  +577.172, Z    +0.000, E1   +75.843, E3 +99557.467}
SPL {X  -159.895, Y  +349.775, Z    +0.000, E1   +76.042, E3 +99649.133}
ENDSPLINE

SPLINE
SPL {X  -160.357, Y  +352.285, Z    +0.000, E1   +74.783, E3 +99662.071}
ENDSPLINE

SPLINE
SPL {X  -145.737, Y  +307.897, Z    +0.000, E1   +77.368, E3 +99654.646}
SPL {X  -145.122, Y  +306.676, Z    +0.000, E1   +76.360, E3 +99665.999}
ENDSPLINE

SPLINE
SPL {X  -145.186, Y  +306.802, Z    +0.000, E1   +74.850, E3 +99680.352}
ENDSPLINE

SPLINE
SPL {X  -143.742, Y  +304.025, Z    +0.000, E1   +73.644, E3 +99692.407}
SPL {X  -141.993, Y  +300.823, Z    +0.000, E1   +72.659, E3 +99701.979}
SPL {X  -138.166, Y  +294.358, Z    +0.000, E1   +72.281, E3 +99708.440}
SPL {X  -134.385, Y  +288.571, Z    +0.000, E1   +71.826, E3 +99714.704}
SPL {X  -129.872, Y  +282.297, Z    +0.000, E1   +71.229, E3 +99721.874}
SPL {X  -124.448, Y  +275.510, Z    +0.000, E1   +70.509, E3 +99729.247}
SPL {X  -117.513, Y  +267.801, Z    +0.000, E1   +72.197, E3 +99726.830}
SPL {X   -63.140, Y  +230.421, Z    +0.000, E1   +55.875, E3 +99896.268}
ENDSPLINE

SPLINE
SPL {X  -130.329, Y  +282.905, Z    +0.000, E1   +55.659, E3 +100054.604}
SPL {X  -150.766, Y  +319.018, Z    +0.000, E1   +45.408, E3 +100063.097}
SPL {X  -157.479, Y  +339.138, Z    +0.000, E1   +35.556, E3 +100064.532}
SPL {X  -160.994, Y  +356.185, Z    +0.000, E1   +24.373, E3 +100066.578}
SPL {X  -162.352, Y  +368.168, Z    +0.000, E1   +14.282, E3 +100066.631}
SPL {X  -162.808, Y  +378.562, Z    +0.000, E1    +4.298, E3 +100066.563}
SPL {X  -162.820, Y  +382.500, Z    +0.000, E1    +0.000, E3 +100066.136}
SPL {X  -162.820, Y  +383.794, Z    +0.000, E1    -2.626, E3 +100065.877}
SPL {X  -162.820, Y  +387.647, Z    +0.000, E1   -11.488, E3 +100065.880}
SPL {X  -162.820, Y  +393.007, Z    +0.000, E1   -25.093, E3 +100065.838}
SPL {X  -162.820, Y  +400.636, Z    +0.000, E1   -41.711, E3 +100065.888}
SPL {X  -162.820, Y  +414.705, Z    +0.000, E1   -61.052, E3 +100065.474}
SPL {X  -162.820, Y  +466.149, Z    +0.000, E1   -74.732, E3 +100075.470}
SPL {X  -160.066, Y  +703.318, Z    +0.000, E1   -76.774, E3 +100160.318}
ENDSPLINE

SPLINE
SPL {X  -161.105, Y  +697.069, Z    +0.000, E1   -74.557, E3 +100181.932}
ENDSPLINE

SPLINE
SPL {X  -159.270, Y  +707.314, Z    +0.000, E1   -74.359, E3 +100189.956}
SPL {X  -156.868, Y  +717.123, Z    +0.000, E1   -74.182, E3 +100197.462}
SPL {X  -153.226, Y  +728.564, Z    +0.000, E1   -73.755, E3 +100208.470}
SPL {X  -149.090, Y  +738.941, Z    +0.000, E1   -73.348, E3 +100218.043}
SPL {X  -145.714, Y  +746.149, Z    +0.000, E1   -72.951, E3 +100225.630}
SPL {X  -140.946, Y  +755.015, Z    +0.000, E1   -72.452, E3 +100234.733}
SPL {X  -136.902, Y  +761.638, Z    +0.000, E1   -71.857, E3 +100242.600}
SPL {X  -133.350, Y  +766.925, Z    +0.000, E1   -71.498, E3 +100247.920}
SPL {X  -129.687, Y  +771.946, Z    +0.000, E1   -71.061, E3 +100253.286}
SPL {X  -126.374, Y  +776.164, Z    +0.000, E1   -70.494, E3 +100258.540}
SPL {X  -123.763, Y  +779.297, Z    +0.000, E1   -70.128, E3 +100261.916}
SPL {X  -119.350, Y  +784.252, Z    +0.000, E1   -71.016, E3 +100261.116}
SPL {X   -61.593, Y  +824.220, Z    +0.000, E1   -55.970, E3 +100427.431}
ENDSPLINE

SPLINE
SPL {X  -131.598, Y  +769.376, Z    +0.000, E1   -56.871, E3 +100593.703}
SPL {X  -152.760, Y  +729.846, Z    +0.000, E1   -44.713, E3 +100600.756}
SPL {X  -158.868, Y  +709.157, Z    +0.000, E1   -33.466, E3 +100601.957}
SPL {X  -161.987, Y  +689.949, Z    +0.000, E1   -18.777, E3 +100602.918}
SPL {X  -162.743, Y  +678.515, Z    +0.000, E1    -7.658, E3 +100602.913}
SPL {X  -162.820, Y  +671.588, Z    +0.000, E1    -0.190, E3 +100602.459}
SPL {X  -162.820, Y  +669.410, Z    +0.000, E1    +4.515, E3 +100602.198}
SPL {X  -162.820, Y  +664.781, Z    +0.000, E1   +16.411, E3 +100602.194}
SPL {X  -162.820, Y  +659.650, Z    +0.000, E1   +29.778, E3 +100602.204}
SPL {X  -162.820, Y  +654.031, Z    +0.000, E1   +42.449, E3 +100602.117}
SPL {X  -162.820, Y  +647.611, Z    +0.000, E1   +52.483, E3 +100602.648}
SPL {X  -162.820, Y  +637.134, Z    +0.000, E1   +65.232, E3 +100600.896}
SPL {X  -162.820, Y  +616.721, Z    +0.000, E1   +72.273, E3 +100604.630}
SPL {X  -162.820, Y  +577.172, Z    +0.000, E1   +75.843, E3 +100614.610}
SPL {X  -159.895, Y  +349.775, Z    +0.000, E1   +76.042, E3 +100706.276}
ENDSPLINE

SPLINE
SPL {X  -160.357, Y  +352.285, Z    +0.000, E1   +74.783, E3 +100719.214}
ENDSPLINE

SPLINE
SPL {X  -145.737, Y  +307.897, Z    +0.000, E1   +77.368, E3 +100711.789}
SPL {X  -145.122, Y  +306.676, Z    +0.000, E1   +76.360, E3 +100723.142}
ENDSPLINE

SPLINE
SPL {X  -145.186, Y  +306.802, Z    +0.000, E1   +74.850, E3 +100737.495}
ENDSPLINE

SPLINE
SPL {X  -143.742, Y  +304.025, Z    +0.000, E1   +73.644, E3 +100749.550}
SPL {X  -141.993, Y  +300.823, Z    +0.000, E1   +72.659, E3 +100759.122}
SPL {X  -138.166, Y  +294.358, Z    +0.000, E1   +72.281, E3 +100765.583}
SPL {X  -134.385, Y  +288.571, Z    +0.000, E1   +71.826, E3 +100771.847}
SPL {X  -129.872, Y  +282.297, Z    +0.000, E1   +71.229, E3 +100779.017}
SPL {X  -124.448, Y  +275.510, Z    +0.000, E1   +70.509, E3 +100786.390}
SPL {X  -117.513, Y  +267.801, Z    +0.000, E1   +72.197, E3 +100783.972}
SPL {X   -63.140, Y  +230.421, Z    +0.000, E1   +55.875, E3 +100953.411}
ENDSPLINE

SPLINE
SPL {X  -130.329, Y  +282.905, Z    +0.000, E1   +55.659, E3 +101111.747}
SPL {X  -150.766, Y  +319.018, Z    +0.000, E1   +45.408, E3 +101120.240}
SPL {X  -157.479, Y  +339.138, Z    +0.000, E1   +35.556, E3 +101121.675}
SPL {X  -160.994, Y  +356.185, Z    +0.000, E1   +24.373, E3 +101123.721}
SPL {X  -162.352, Y  +368.168, Z    +0.000, E1   +14.282, E3 +101123.774}
SPL {X  -162.808, Y  +378.562, Z    +0.000, E1    +4.298, E3 +101123.706}
SPL {X  -162.820, Y  +382.500, Z    +0.000, E1    +0.000, E3 +101123.278}
SPL {X  -162.820, Y  +383.794, Z    +0.000, E1    -2.626, E3 +101123.019}
SPL {X  -162.820, Y  +387.647, Z    +0.000, E1   -11.488, E3 +101123.023}
SPL {X  -162.820, Y  +393.007, Z    +0.000, E1   -25.093, E3 +101122.981}
SPL {X  -162.820, Y  +400.636, Z    +0.000, E1   -41.711, E3 +101123.030}
SPL {X  -162.820, Y  +414.705, Z    +0.000, E1   -61.052, E3 +101122.617}
SPL {X  -162.820, Y  +466.149, Z    +0.000, E1   -74.732, E3 +101132.613}
SPL {X  -160.066, Y  +703.318, Z    +0.000, E1   -76.774, E3 +101217.461}
ENDSPLINE

SPLINE
SPL {X  -161.105, Y  +697.069, Z    +0.000, E1   -74.557, E3 +101239.075}
ENDSPLINE

SPLINE
SPL {X  -159.270, Y  +707.314, Z    +0.000, E1   -74.359, E3 +101247.099}
SPL {X  -156.868, Y  +717.123, Z    +0.000, E1   -74.182, E3 +101254.605}
SPL {X  -153.226, Y  +728.564, Z    +0.000, E1   -73.755, E3 +101265.613}
SPL {X  -149.090, Y  +738.941, Z    +0.000, E1   -73.348, E3 +101275.186}
SPL {X  -145.714, Y  +746.149, Z    +0.000, E1   -72.951, E3 +101282.773}
SPL {X  -140.946, Y  +755.015, Z    +0.000, E1   -72.452, E3 +101291.876}
SPL {X  -136.902, Y  +761.638, Z    +0.000, E1   -71.857, E3 +101299.743}
SPL {X  -133.350, Y  +766.925, Z    +0.000, E1   -71.498, E3 +101305.063}
SPL {X  -129.687, Y  +771.946, Z    +0.000, E1   -71.061, E3 +101310.429}
SPL {X  -126.374, Y  +776.164, Z    +0.000, E1   -70.494, E3 +101315.683}
SPL {X  -123.763, Y  +779.297, Z    +0.000, E1   -70.128, E3 +101319.059}
SPL {X  -119.350, Y  +784.252, Z    +0.000, E1   -71.016, E3 +101318.259}
SPL {X   -61.593, Y  +824.220, Z    +0.000, E1   -55.970, E3 +101484.574}
ENDSPLINE

SPLINE
SPL {X  -131.598, Y  +769.376, Z    +0.000, E1   -56.871, E3 +101650.846}
SPL {X  -152.760, Y  +729.846, Z    +0.000, E1   -44.713, E3 +101657.898}
SPL {X  -158.868, Y  +709.157, Z    +0.000, E1   -33.466, E3 +101659.099}
SPL {X  -161.987, Y  +689.949, Z    +0.000, E1   -18.777, E3 +101660.061}
SPL {X  -162.743, Y  +678.515, Z    +0.000, E1    -7.658, E3 +101660.056}
SPL {X  -162.820, Y  +671.588, Z    +0.000, E1    -0.190, E3 +101659.602}
SPL {X  -162.820, Y  +669.410, Z    +0.000, E1    +4.515, E3 +101659.341}
SPL {X  -162.820, Y  +664.781, Z    +0.000, E1   +16.411, E3 +101659.337}
SPL {X  -162.820, Y  +659.650, Z    +0.000, E1   +29.778, E3 +101659.346}
SPL {X  -162.820, Y  +654.031, Z    +0.000, E1   +42.449, E3 +101659.260}
SPL {X  -162.820, Y  +647.611, Z    +0.000, E1   +52.483, E3 +101659.791}
SPL {X  -162.820, Y  +637.134, Z    +0.000, E1   +65.232, E3 +101658.039}
SPL {X  -162.820, Y  +616.721, Z    +0.000, E1   +72.273, E3 +101661.773}
SPL {X  -162.820, Y  +577.172, Z    +0.000, E1   +75.843, E3 +101671.753}
SPL {X  -159.895, Y  +349.775, Z    +0.000, E1   +76.042, E3 +101763.419}
ENDSPLINE

SPLINE
SPL {X  -160.357, Y  +352.285, Z    +0.000, E1   +74.783, E3 +101776.357}
ENDSPLINE

SPLINE
SPL {X  -145.737, Y  +307.897, Z    +0.000, E1   +77.368, E3 +101768.932}
SPL {X  -145.122, Y  +306.676, Z    +0.000, E1   +76.360, E3 +101780.285}
ENDSPLINE

SPLINE
SPL {X  -145.186, Y  +306.802, Z    +0.000, E1   +74.850, E3 +101794.638}
ENDSPLINE

SPLINE
SPL {X  -143.742, Y  +304.025, Z    +0.000, E1   +73.644, E3 +101806.692}
SPL {X  -141.993, Y  +300.823, Z    +0.000, E1   +72.659, E3 +101816.265}
SPL {X  -138.166, Y  +294.358, Z    +0.000, E1   +72.281, E3 +101822.726}
SPL {X  -134.385, Y  +288.571, Z    +0.000, E1   +71.826, E3 +101828.990}
SPL {X  -129.872, Y  +282.297, Z    +0.000, E1   +71.229, E3 +101836.160}
SPL {X  -124.448, Y  +275.510, Z    +0.000, E1   +70.509, E3 +101843.533}
SPL {X  -117.513, Y  +267.801, Z    +0.000, E1   +72.197, E3 +101841.115}
SPL {X   -63.140, Y  +230.421, Z    +0.000, E1   +55.875, E3 +102010.554}
ENDSPLINE

SPLINE
SPL {X  -130.329, Y  +282.905, Z    +0.000, E1   +55.659, E3 +102168.890}
SPL {X  -150.766, Y  +319.018, Z    +0.000, E1   +45.408, E3 +102177.383}
SPL {X  -157.479, Y  +339.138, Z    +0.000, E1   +35.556, E3 +102178.818}
SPL {X  -160.994, Y  +356.185, Z    +0.000, E1   +24.373, E3 +102180.864}
SPL {X  -162.352, Y  +368.168, Z    +0.000, E1   +14.282, E3 +102180.917}
SPL {X  -162.808, Y  +378.562, Z    +0.000, E1    +4.298, E3 +102180.848}
SPL {X  -162.820, Y  +382.500, Z    +0.000, E1    +0.000, E3 +102180.421}
SPL {X  -162.820, Y  +383.794, Z    +0.000, E1    -2.626, E3 +102180.162}
SPL {X  -162.820, Y  +387.647, Z    +0.000, E1   -11.488, E3 +102180.166}
SPL {X  -162.820, Y  +393.007, Z    +0.000, E1   -25.093, E3 +102180.124}
SPL {X  -162.820, Y  +400.636, Z    +0.000, E1   -41.711, E3 +102180.173}
SPL {X  -162.820, Y  +414.705, Z    +0.000, E1   -61.052, E3 +102179.760}
SPL {X  -162.820, Y  +466.149, Z    +0.000, E1   -74.732, E3 +102189.756}
SPL {X  -160.722, Y  +699.554, Z    +0.000, E1   -75.485, E3 +102287.166}
SPL {X  -159.966, Y  +703.854, Z    +0.000, E1   -74.386, E3 +102302.069}
SPL {X  -156.868, Y  +717.123, Z    +0.000, E1   -74.182, E3 +102311.747}
SPL {X  -154.373, Y  +725.261, Z    +0.000, E1   -73.879, E3 +102319.457}
SPL {X  -152.060, Y  +731.708, Z    +0.000, E1   -73.572, E3 +102326.105}
SPL {X  -149.090, Y  +738.941, Z    +0.000, E1   -73.348, E3 +102332.329}
SPL {X  -145.714, Y  +746.149, Z    +0.000, E1   -72.951, E3 +102339.916}
SPL {X  -142.592, Y  +752.100, Z    +0.000, E1   -72.554, E3 +102346.449}
SPL {X  -139.608, Y  +757.285, Z    +0.000, E1   -72.326, E3 +102351.118}
SPL {X  -136.902, Y  +761.638, Z    +0.000, E1   -71.857, E3 +102356.886}
SPL {X  -133.350, Y  +766.925, Z    +0.000, E1   -71.498, E3 +102362.206}
SPL {X  -129.687, Y  +771.946, Z    +0.000, E1   -71.061, E3 +102367.572}
SPL {X  -126.374, Y  +776.164, Z    +0.000, E1   -70.494, E3 +102372.826}
SPL {X  -122.717, Y  +780.508, Z    +0.000, E1   -70.361, E3 +102375.863}
SPL {X  -114.093, Y  +789.660, Z    +0.000, E1   -71.634, E3 +102375.881}
SPL {X   -61.593, Y  +824.220, Z    +0.000, E1   -55.970, E3 +102541.717}
ENDSPLINE

SPLINE
SPL {X  -131.598, Y  +769.376, Z    +0.000, E1   -56.871, E3 +102707.989}
SPL {X  -152.760, Y  +729.846, Z    +0.000, E1   -44.713, E3 +102715.041}
SPL {X  -158.868, Y  +709.157, Z    +0.000, E1   -33.466, E3 +102716.242}
SPL {X  -161.987, Y  +689.949, Z    +0.000, E1   -18.777, E3 +102717.203}
SPL {X  -162.803, Y  +675.860, Z    +0.000, E1    -4.958, E3 +102717.186}
SPL {X  -162.820, Y  +671.500, Z    +0.000, E1    +0.000, E3 +102716.722}
SPL {X  -162.820, Y  +669.410, Z    +0.000, E1    +4.515, E3 +102716.484}
SPL {X  -162.820, Y  +664.781, Z    +0.000, E1   +16.411, E3 +102716.480}
SPL {X  -162.820, Y  +659.650, Z    +0.000, E1   +29.778, E3 +102716.489}
SPL {X  -162.820, Y  +651.175, Z    +0.000, E1   +47.162, E3 +102716.639}
SPL {X  -162.820, Y  +637.134, Z    +0.000, E1   +65.232, E3 +102715.181}
SPL {X  -162.820, Y  +616.721, Z    +0.000, E1   +72.273, E3 +102718.915}
SPL {X  -162.820, Y  +577.172, Z    +0.000, E1   +75.843, E3 +102728.896}
SPL {X  -159.895, Y  +349.775, Z    +0.000, E1   +76.042, E3 +102820.562}
ENDSPLINE

SPLINE
SPL {X  -160.357, Y  +352.285, Z    +0.000, E1   +74.783, E3 +102833.500}
ENDSPLINE

SPLINE
SPL {X  -145.737, Y  +307.897, Z    +0.000, E1   +77.368, E3 +102826.075}
SPL {X  -145.329, Y  +307.084, Z    +0.000, E1   +76.571, E3 +102834.911}
ENDSPLINE

SPLINE
SPL {X  -145.355, Y  +307.136, Z    +0.000, E1   +75.607, E3 +102844.435}
ENDSPLINE

SPLINE
SPL {X  -144.515, Y  +305.495, Z    +0.000, E1   +74.543, E3 +102855.244}
SPL {X  -143.690, Y  +303.925, Z    +0.000, E1   +73.372, E3 +102865.983}
SPL {X  -141.993, Y  +300.823, Z    +0.000, E1   +72.659, E3 +102873.408}
SPL {X  -138.166, Y  +294.358, Z    +0.000, E1   +72.281, E3 +102879.869}
SPL {X  -134.385, Y  +288.571, Z    +0.000, E1   +71.826, E3 +102886.132}
SPL {X  -129.872, Y  +282.297, Z    +0.000, E1   +71.229, E3 +102893.303}
SPL {X  -124.448, Y  +275.510, Z    +0.000, E1   +70.509, E3 +102900.675}
SPL {X  -117.513, Y  +267.801, Z    +0.000, E1   +72.197, E3 +102898.258}
SPL {X   -63.140, Y  +230.421, Z    +0.000, E1   +55.875, E3 +103067.697}
ENDSPLINE

SPLINE
SPL {X  -130.329, Y  +282.905, Z    +0.000, E1   +55.659, E3 +103226.033}
SPL {X  -150.766, Y  +319.018, Z    +0.000, E1   +45.408, E3 +103234.525}
SPL {X  -157.479, Y  +339.138, Z    +0.000, E1   +35.556, E3 +103235.961}
SPL {X  -160.994, Y  +356.185, Z    +0.000, E1   +24.373, E3 +103238.007}
SPL {X  -162.352, Y  +368.168, Z    +0.000, E1   +14.282, E3 +103238.059}
SPL {X  -162.808, Y  +378.562, Z    +0.000, E1    +4.298, E3 +103237.991}
SPL {X  -162.820, Y  +382.500, Z    +0.000, E1    +0.000, E3 +103237.564}
SPL {X  -162.820, Y  +384.915, Z    +0.000, E1    -4.894, E3 +103237.277}
SPL {X  -162.820, Y  +388.986, Z    +0.000, E1   -15.047, E3 +103237.375}
SPL {X  -162.820, Y  +394.732, Z    +0.000, E1   -28.992, E3 +103237.227}
SPL {X  -162.820, Y  +403.075, Z    +0.000, E1   -46.096, E3 +103237.456}
SPL {X  -162.820, Y  +414.705, Z    +0.000, E1   -61.052, E3 +103236.903}
SPL {X  -162.820, Y  +466.149, Z    +0.000, E1   -74.732, E3 +103246.899}
SPL {X  -160.722, Y  +699.554, Z    +0.000, E1   -75.485, E3 +103344.309}
SPL {X  -159.966, Y  +703.854, Z    +0.000, E1   -74.386, E3 +103359.212}
SPL {X  -156.868, Y  +717.123, Z    +0.000, E1   -74.182, E3 +103368.890}
SPL {X  -153.226, Y  +728.564, Z    +0.000, E1   -73.755, E3 +103379.898}
SPL {X  -149.090, Y  +738.941, Z    +0.000, E1   -73.348, E3 +103389.472}
SPL {X  -145.714, Y  +746.149, Z    +0.000, E1   -72.951, E3 +103397.059}
SPL {X  -140.946, Y  +755.015, Z    +0.000, E1   -72.452, E3 +103406.162}
SPL {X  -136.902, Y  +761.638, Z    +0.000, E1   -71.857, E3 +103414.028}
SPL {X  -133.350, Y  +766.925, Z    +0.000, E1   -71.498, E3 +103419.349}
SPL {X  -129.687, Y  +771.946, Z    +0.000, E1   -71.061, E3 +103424.715}
SPL {X  -126.374, Y  +776.164, Z    +0.000, E1   -70.494, E3 +103429.968}
SPL {X  -122.717, Y  +780.508, Z    +0.000, E1   -70.361, E3 +103433.006}
SPL {X  -114.093, Y  +789.660, Z    +0.000, E1   -71.634, E3 +103433.024}
SPL {X   -61.593, Y  +824.220, Z    +0.000, E1   -55.970, E3 +103598.860}
ENDSPLINE

SPLINE
SPL {X  -131.598, Y  +769.376, Z    +0.000, E1   -56.871, E3 +103765.132}
SPL {X  -152.760, Y  +729.846, Z    +0.000, E1   -44.713, E3 +103772.184}
SPL {X  -158.868, Y  +709.157, Z    +0.000, E1   -33.466, E3 +103773.385}
SPL {X  -161.987, Y  +689.949, Z    +0.000, E1   -18.777, E3 +103774.346}
SPL {X  -162.803, Y  +675.860, Z    +0.000, E1    -4.958, E3 +103774.328}
SPL {X  -162.820, Y  +671.500, Z    +0.000, E1    +0.000, E3 +103773.865}
SPL {X  -162.820, Y  +669.410, Z    +0.000, E1    +4.515, E3 +103773.627}
SPL {X  -162.820, Y  +664.781, Z    +0.000, E1   +16.411, E3 +103773.622}
SPL {X  -162.820, Y  +659.650, Z    +0.000, E1   +29.778, E3 +103773.632}
SPL {X  -162.820, Y  +651.175, Z    +0.000, E1   +47.162, E3 +103773.782}
SPL {X  -162.820, Y  +637.134, Z    +0.000, E1   +65.232, E3 +103772.324}
SPL {X  -162.820, Y  +616.721, Z    +0.000, E1   +72.273, E3 +103776.058}
SPL {X  -162.820, Y  +577.172, Z    +0.000, E1   +75.843, E3 +103786.039}
SPL {X  -159.895, Y  +349.775, Z    +0.000, E1   +76.042, E3 +103877.705}
ENDSPLINE

SPLINE
SPL {X  -160.357, Y  +352.285, Z    +0.000, E1   +74.783, E3 +103890.642}
ENDSPLINE

SPLINE
SPL {X  -145.737, Y  +307.897, Z    +0.000, E1   +77.368, E3 +103883.218}
SPL {X  -145.329, Y  +307.084, Z    +0.000, E1   +76.571, E3 +103892.054}
ENDSPLINE

SPLINE
SPL {X  -145.355, Y  +307.136, Z    +0.000, E1   +75.607, E3 +103901.578}
ENDSPLINE

SPLINE
SPL {X  -144.515, Y  +305.495, Z    +0.000, E1   +74.543, E3 +103912.387}
SPL {X  -143.690, Y  +303.925, Z    +0.000, E1   +73.372, E3 +103923.126}
SPL {X  -141.993, Y  +300.823, Z    +0.000, E1   +72.659, E3 +103930.551}
SPL {X  -138.166, Y  +294.358, Z    +0.000, E1   +72.281, E3 +103937.012}
SPL {X  -134.385, Y  +288.571, Z    +0.000, E1   +71.826, E3 +103943.275}
SPL {X  -130.773, Y  +283.501, Z    +0.000, E1   +71.398, E3 +103948.700}
SPL {X  -126.922, Y  +278.513, Z    +0.000, E1   +70.767, E3 +103954.854}
SPL {X  -123.520, Y  +274.419, Z    +0.000, E1   +70.342, E3 +103959.052}
SPL {X  -117.513, Y  +267.801, Z    +0.000, E1   +72.197, E3 +103955.401}
SPL {X   -63.140, Y  +230.421, Z    +0.000, E1   +55.875, E3 +104124.840}
ENDSPLINE

SPLINE
SPL {X  -130.329, Y  +282.905, Z    +0.000, E1   +55.659, E3 +104283.176}
SPL {X  -154.728, Y  +329.807, Z    +0.000, E1   +40.640, E3 +104292.557}
SPL {X  -160.994, Y  +356.185, Z    +0.000, E1   +24.373, E3 +104295.150}
SPL {X  -162.637, Y  +372.778, Z    +0.000, E1   +10.098, E3 +104295.170}
SPL {X  -162.820, Y  +382.748, Z    +0.000, E1    -0.178, E3 +104294.662}
SPL {X  -162.820, Y  +387.647, Z    +0.000, E1   -11.488, E3 +104294.451}
SPL {X  -162.820, Y  +393.007, Z    +0.000, E1   -25.093, E3 +104294.409}
SPL {X  -162.820, Y  +400.636, Z    +0.000, E1   -41.711, E3 +104294.459}
SPL {X  -162.820, Y  +414.705, Z    +0.000, E1   -61.052, E3 +104294.046}
SPL {X  -162.820, Y  +466.149, Z    +0.000, E1   -74.732, E3 +104304.042}
SPL {X  -160.066, Y  +703.318, Z    +0.000, E1   -76.774, E3 +104388.889}
ENDSPLINE

SPLINE
SPL {X  -161.105, Y  +697.069, Z    +0.000, E1   -74.557, E3 +104410.503}
ENDSPLINE

SPLINE
SPL {X  -159.270, Y  +707.314, Z    +0.000, E1   -74.359, E3 +104418.527}
SPL {X  -156.868, Y  +717.123, Z    +0.000, E1   -74.182, E3 +104426.033}
SPL {X  -154.373, Y  +725.261, Z    +0.000, E1   -73.879, E3 +104433.743}
SPL {X  -152.060, Y  +731.708, Z    +0.000, E1   -73.572, E3 +104440.391}
SPL {X  -149.090, Y  +738.941, Z    +0.000, E1   -73.348, E3 +104446.615}
SPL {X  -145.714, Y  +746.149, Z    +0.000, E1   -72.951, E3 +104454.202}
SPL {X  -140.946, Y  +755.015, Z    +0.000, E1   -72.452, E3 +104463.305}
SPL {X  -136.902, Y  +761.638, Z    +0.000, E1   -71.857, E3 +104471.171}
SPL {X  -133.350, Y  +766.925, Z    +0.000, E1   -71.498, E3 +104476.492}
SPL {X  -129.687, Y  +771.946, Z    +0.000, E1   -71.061, E3 +104481.858}
SPL {X  -126.374, Y  +776.164, Z    +0.000, E1   -70.494, E3 +104487.111}
SPL {X  -122.717, Y  +780.508, Z    +0.000, E1   -70.361, E3 +104490.149}
SPL {X  -114.093, Y  +789.660, Z    +0.000, E1   -71.634, E3 +104490.167}
SPL {X   -61.795, Y  +824.138, Z    +0.000, E1   -56.629, E3 +104635.834}
ENDSPLINE

SPLINE
SPL {X  -113.687, Y  +790.058, Z    +0.000, E1   -59.721, E3 +104812.582}
SPL {X  -139.151, Y  +758.042, Z    +0.000, E1   -54.091, E3 +104824.141}
SPL {X  -152.760, Y  +729.846, Z    +0.000, E1   -44.713, E3 +104829.327}
SPL {X  -158.868, Y  +709.157, Z    +0.000, E1   -33.466, E3 +104830.528}
SPL {X  -161.987, Y  +689.949, Z    +0.000, E1   -18.777, E3 +104831.489}
SPL {X  -162.743, Y  +678.515, Z    +0.000, E1    -7.658, E3 +104831.484}
SPL {X  -162.820, Y  +671.380, Z    +0.000, E1    +0.035, E3 +104830.989}
SPL {X  -162.820, Y  +668.318, Z    +0.000, E1    +7.404, E3 +104830.726}
SPL {X  -162.820, Y  +664.781, Z    +0.000, E1   +16.411, E3 +104830.765}
SPL {X  -162.820, Y  +659.650, Z    +0.000, E1   +29.778, E3 +104830.775}
SPL {X  -162.820, Y  +651.175, Z    +0.000, E1   +47.162, E3 +104830.925}
SPL {X  -162.820, Y  +633.243, Z    +0.000, E1   +67.111, E3 +104830.180}
SPL {X  -162.820, Y  +577.172, Z    +0.000, E1   +75.843, E3 +104843.181}
SPL {X  -159.895, Y  +349.775, Z    +0.000, E1   +76.042, E3 +104934.848}
ENDSPLINE

SPLINE
SPL {X  -160.357, Y  +352.285, Z    +0.000, E1   +74.783, E3 +104947.785}
ENDSPLINE

SPLINE
SPL {X  -145.737, Y  +307.897, Z    +0.000, E1   +77.368, E3 +104940.361}
SPL {X  -145.329, Y  +307.084, Z    +0.000, E1   +76.571, E3 +104949.197}
ENDSPLINE

SPLINE
SPL {X  -145.355, Y  +307.136, Z    +0.000, E1   +75.607, E3 +104958.721}
ENDSPLINE

